KUKA KRL program: f1_Kuka_APT205T03S05.SRC

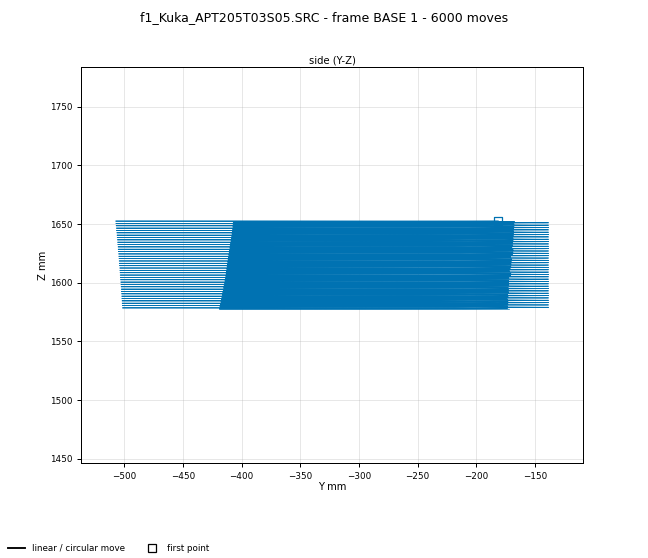
[picture p0: tool path of f1_Kuka_APT205T03S05.SRC in frame BASE 1, 6000 of 6001 moves have a stored position in this frame; points joined in program order, loops and branches not executed]
&ACCESS RVP
&REL 2
&PARAM TEMPLATE = C:\KRC\Roboter\Template\vorgabe
&PARAM EDITMASK = *
DEF f1_Kuka_APT205T03S05()


;FOLD INI;%{PE}%V3.2.0,%MKUKATPBASIS,%CINIT,%VCOMMON,%P
  ;FOLD BAS INI;%{E}%V3.2.0,%MKUKATPBASIS,%CINIT,%VINIT,%P
    GLOBAL INTERRUPT DECL 3 WHEN $STOPMESS==TRUE DO IR_STOPM ( )
    INTERRUPT ON 3
    BAS (#INITMOV,0 )
  ;ENDFOLD (BAS INI)
  ;FOLD USER INI;%{E}%V3.2.0,%MKUKATPUSER,%CINIT,%VINIT,%P
    ;Make your modifications here
  ;ENDFOLD (USER INI)
;ENDFOLD (INI)


;*** Make Null PTP Move
  PTP $pos_act

;*** Auto Load The Correct TOOL Data
  $tool=tool_data[3]

;*** Auto Load The Correct BASE Data
  $base=base_data[1]

  $ADVANCE = 5

;*** Restate Last Velocity
MMPM(30000.0)
SetRPM(6000)
LIN {X -0.097,Y -181.135,Z 1652.752,A 0.000,B 0.000,C 90.000,E1 135.405} C_DIS
LIN {X 0.030,Y -186.585,Z 1652.733,A 0.000,B 0.000,C 90.000,E1 132.000} C_DIS
LIN {X -0.021,Y -191.197,Z 1652.719,A 0.000,B 0.000,C 90.000,E1 129.519} C_DIS
LIN {X 0.024,Y -197.007,Z 1652.701,A 0.000,B 0.000,C 90.000,E1 126.217} C_DIS
LIN {X -0.058,Y -200.276,Z 1652.692,A 0.000,B 0.000,C 90.000,E1 124.612} C_DIS
LIN {X 0.005,Y -207.052,Z 1652.672,A 0.000,B 0.000,C 90.000,E1 120.924} C_DIS
LIN {X -0.045,Y -328.099,Z 1652.672,A 0.000,B 0.000,C 90.000,E1 120.924} C_DIS
LIN {X -0.152,Y -329.288,Z 1652.672,A 0.000,B 0.000,C 90.000,E1 120.924} C_DIS
LIN {X 0.100,Y -333.426,Z 1652.671,A 0.000,B 0.000,C 90.000,E1 120.718} C_DIS
LIN {X -0.104,Y -335.740,Z 1652.670,A 0.000,B 0.000,C 90.000,E1 120.590} C_DIS
LIN {X 0.166,Y -339.608,Z 1652.667,A 0.000,B 0.000,C 90.000,E1 120.129} C_DIS
LIN {X -0.040,Y -341.484,Z 1652.666,A 0.000,B 0.000,C 90.000,E1 119.873} C_DIS
LIN {X -0.079,Y -342.956,Z 1652.664,A 0.000,B 0.000,C 90.000,E1 119.589} C_DIS
LIN {X 0.037,Y -355.225,Z 1652.649,A 0.000,B 0.000,C 90.000,E1 116.821} C_DIS
LIN {X 0.029,Y -368.954,Z 1652.634,A 0.000,B 0.000,C 90.000,E1 114.131} C_DIS
LIN {X 0.163,Y -382.488,Z 1652.621,A 0.000,B 0.000,C 90.000,E1 111.770} C_DIS
LIN {X -0.003,Y -397.372,Z 1652.608,A 0.000,B 0.000,C 90.000,E1 109.504} C_DIS
LIN {X -0.071,Y -413.709,Z 1652.596,A 0.000,B 0.000,C 90.000,E1 107.275} C_DIS
LIN {X 0.146,Y -431.611,Z 1652.584,A 0.000,B 0.000,C 90.000,E1 105.064} C_DIS
LIN {X 0.171,Y -451.069,Z 1652.572,A 0.000,B 0.000,C 90.000,E1 102.952} C_DIS
LIN {X 0.102,Y -471.266,Z 1652.561,A 0.000,B 0.000,C 90.000,E1 101.007} C_DIS
LIN {X -0.176,Y -494.592,Z 1652.550,A 0.000,B 0.000,C 90.000,E1 99.029} C_DIS
LIN {X 0.166,Y -499.819,Z 1652.548,A 0.000,B 0.000,C 90.000,E1 98.568} C_DIS
LIN {X -0.174,Y -501.889,Z 1652.547,A 0.000,B 0.000,C 90.000,E1 98.398} C_DIS
LIN {X -0.238,Y -503.694,Z 1652.545,A 0.000,B 0.000,C 90.000,E1 98.163} C_DIS
LIN {X 0.198,Y -505.046,Z 1652.544,A 0.000,B 0.000,C 90.000,E1 97.871} C_DIS
LIN {X 0.003,Y -506.730,Z 1652.541,A 0.000,B 0.000,C 90.000,E1 97.409} C_DIS
LIN {X -0.185,Y -507.309,Z 1652.538,A 0.000,B 0.000,C 90.000,E1 96.947} C_DIS
LIN {X 0.141,Y -506.879,Z 1652.536,A 0.000,B 0.000,C 90.000,E1 96.429} C_DIS
LIN {X -0.035,Y -505.372,Z 1652.533,A 0.000,B 0.000,C 90.000,E1 95.967} C_DIS
LIN {X -0.149,Y -504.130,Z 1652.532,A 0.000,B 0.000,C 90.000,E1 95.739} C_DIS
LIN {X 0.200,Y -493.883,Z 1652.524,A 0.000,B 0.000,C 90.000,E1 94.245} C_DIS
LIN {X 0.044,Y -479.975,Z 1652.513,A 0.000,B 0.000,C 90.000,E1 92.293} C_DIS
LIN {X -0.050,Y -469.373,Z 1652.504,A 0.000,B 0.000,C 90.000,E1 90.802} C_DIS
LIN {X 0.134,Y -458.498,Z 1652.496,A 0.000,B 0.000,C 90.000,E1 89.255} C_DIS
LIN {X 0.134,Y -447.360,Z 1652.487,A 0.000,B 0.000,C 90.000,E1 87.707} C_DIS
LIN {X 0.215,Y -437.747,Z 1652.480,A 0.000,B 0.000,C 90.000,E1 86.388} C_DIS
LIN {X 0.171,Y -422.149,Z 1652.468,A 0.000,B 0.000,C 90.000,E1 84.261} C_DIS
LIN {X 0.124,Y -401.321,Z 1652.452,A 0.000,B 0.000,C 90.000,E1 81.254} C_DIS
LIN {X -0.095,Y -383.647,Z 1652.436,A 0.000,B 0.000,C 90.000,E1 78.465} C_DIS
LIN {X 0.146,Y -370.170,Z 1652.423,A 0.000,B 0.000,C 90.000,E1 76.117} C_DIS
LIN {X -0.154,Y -355.532,Z 1652.408,A 0.000,B 0.000,C 90.000,E1 73.504} C_DIS
LIN {X 0.037,Y -338.619,Z 1652.390,A 0.000,B 0.000,C 90.000,E1 70.134} C_DIS
LIN {X -0.145,Y -324.106,Z 1652.372,A 0.000,B 0.000,C 90.000,E1 67.050} C_DIS
LIN {X 0.007,Y -311.770,Z 1652.356,A 0.000,B 0.000,C 90.000,E1 64.152} C_DIS
LIN {X -0.105,Y -302.362,Z 1652.344,A 0.000,B 0.000,C 90.000,E1 61.897} C_DIS
LIN {X 0.124,Y -294.176,Z 1652.333,A 0.000,B 0.000,C 90.000,E1 59.871} C_DIS
LIN {X 0.086,Y -285.764,Z 1652.322,A 0.000,B 0.000,C 90.000,E1 57.867} C_DIS
LIN {X -0.036,Y -277.148,Z 1652.310,A 0.000,B 0.000,C 90.000,E1 55.849} C_DIS
LIN {X -0.016,Y -264.307,Z 1652.293,A 0.000,B 0.000,C 90.000,E1 52.718} C_DIS
LIN {X -0.141,Y -252.123,Z 1652.275,A 0.000,B 0.000,C 90.000,E1 49.542} C_DIS
LIN {X 0.060,Y -240.802,Z 1652.257,A 0.000,B 0.000,C 90.000,E1 46.215} C_DIS
LIN {X 0.093,Y -230.192,Z 1652.238,A 0.000,B 0.000,C 90.000,E1 42.852} C_DIS
LIN {X -0.001,Y -222.452,Z 1652.223,A 0.000,B 0.000,C 90.000,E1 40.216} C_DIS
LIN {X -0.092,Y -214.265,Z 1652.206,A 0.000,B 0.000,C 90.000,E1 37.156} C_DIS
LIN {X 0.005,Y -206.781,Z 1652.189,A 0.000,B 0.000,C 90.000,E1 33.992} C_DIS
LIN {X 0.029,Y -199.997,Z 1652.171,A 0.000,B 0.000,C 90.000,E1 30.797} C_DIS
LIN {X -0.070,Y -193.846,Z 1652.153,A 0.000,B 0.000,C 90.000,E1 27.590} C_DIS
LIN {X 0.025,Y -188.349,Z 1652.135,A 0.000,B 0.000,C 90.000,E1 24.283} C_DIS
LIN {X -0.004,Y -183.536,Z 1652.116,A 0.000,B 0.000,C 90.000,E1 20.972} C_DIS
LIN {X -0.072,Y -179.472,Z 1652.098,A 0.000,B 0.000,C 90.000,E1 17.638} C_DIS
LIN {X 0.069,Y -175.312,Z 1652.074,A 0.000,B 0.000,C 90.000,E1 13.355} C_DIS
LIN {X 0.019,Y -172.038,Z 1652.051,A 0.000,B 0.000,C 90.000,E1 9.095} C_DIS
LIN {X -0.078,Y -169.188,Z 1652.022,A 0.000,B 0.000,C 90.000,E1 3.955} C_DIS
LIN {X 0.014,Y -167.305,Z 1651.973,A 0.000,B 0.000,C 90.000,E1 355.179} C_DIS
LIN {X 0.071,Y -169.078,Z 1651.925,A 0.000,B 0.000,C 90.000,E1 346.464} C_DIS
LIN {X 0.068,Y -172.238,Z 1651.896,A 0.000,B 0.000,C 90.000,E1 341.275} C_DIS
LIN {X 0.041,Y -175.362,Z 1651.877,A 0.000,B 0.000,C 90.000,E1 337.847} C_DIS
LIN {X -0.036,Y -179.335,Z 1651.858,A 0.000,B 0.000,C 90.000,E1 334.460} C_DIS
LIN {X 0.059,Y -184.118,Z 1651.839,A 0.000,B 0.000,C 90.000,E1 331.051} C_DIS
LIN {X -0.040,Y -189.726,Z 1651.821,A 0.000,B 0.000,C 90.000,E1 327.740} C_DIS
LIN {X -0.042,Y -194.546,Z 1651.807,A 0.000,B 0.000,C 90.000,E1 325.261} C_DIS
LIN {X 0.008,Y -201.907,Z 1651.789,A 0.000,B 0.000,C 90.000,E1 321.984} C_DIS
LIN {X 0.018,Y -209.147,Z 1651.773,A 0.000,B 0.000,C 90.000,E1 319.175} C_DIS
LIN {X -0.091,Y -218.598,Z 1651.756,A 0.000,B 0.000,C 90.000,E1 316.053} C_DIS
LIN {X -0.050,Y -227.911,Z 1651.741,A 0.000,B 0.000,C 90.000,E1 313.338} C_DIS
LIN {X 0.015,Y -239.781,Z 1651.724,A 0.000,B 0.000,C 90.000,E1 310.297} C_DIS
LIN {X -0.068,Y -249.776,Z 1651.712,A 0.000,B 0.000,C 90.000,E1 308.096} C_DIS
LIN {X -0.143,Y -259.013,Z 1651.701,A 0.000,B 0.000,C 90.000,E1 306.297} C_DIS
LIN {X -0.036,Y -273.256,Z 1651.688,A 0.000,B 0.000,C 90.000,E1 303.785} C_DIS
LIN {X 0.115,Y -288.938,Z 1651.674,A 0.000,B 0.000,C 90.000,E1 301.337} C_DIS
LIN {X -0.030,Y -310.825,Z 1651.657,A 0.000,B 0.000,C 90.000,E1 298.359} C_DIS
LIN {X 0.020,Y -320.884,Z 1651.650,A 0.000,B 0.000,C 90.000,E1 297.052} C_DIS
LIN {X -0.030,Y -335.600,Z 1651.640,A 0.000,B 0.000,C 90.000,E1 295.155} C_DIS
LIN {X 0.067,Y -350.105,Z 1651.629,A 0.000,B 0.000,C 90.000,E1 293.281} C_DIS
LIN {X 0.115,Y -364.580,Z 1651.619,A 0.000,B 0.000,C 90.000,E1 291.461} C_DIS
LIN {X -0.048,Y -374.011,Z 1651.613,A 0.000,B 0.000,C 90.000,E1 290.301} C_DIS
LIN {X 0.143,Y -380.575,Z 1651.608,A 0.000,B 0.000,C 90.000,E1 289.396} C_DIS
LIN {X 0.032,Y -386.692,Z 1651.603,A 0.000,B 0.000,C 90.000,E1 288.544} C_DIS
LIN {X -0.020,Y -392.189,Z 1651.598,A 0.000,B 0.000,C 90.000,E1 287.692} C_DIS
LIN {X -0.150,Y -396.893,Z 1651.594,A 0.000,B 0.000,C 90.000,E1 286.858} C_DIS
LIN {X 0.156,Y -400.685,Z 1651.589,A 0.000,B 0.000,C 90.000,E1 285.969} C_DIS
LIN {X 0.110,Y -403.624,Z 1651.584,A 0.000,B 0.000,C 90.000,E1 285.134} C_DIS
LIN {X -0.006,Y -405.122,Z 1651.581,A 0.000,B 0.000,C 90.000,E1 284.592} C_DIS
LIN {X 0.179,Y -406.217,Z 1651.578,A 0.000,B 0.000,C 90.000,E1 284.008} C_DIS
LIN {X -0.019,Y -406.894,Z 1651.575,A 0.000,B 0.000,C 90.000,E1 283.480} C_DIS
LIN {X -0.117,Y -407.125,Z 1651.572,A 0.000,B 0.000,C 90.000,E1 282.939} C_DIS
LIN {X 0.090,Y -406.897,Z 1651.569,A 0.000,B 0.000,C 90.000,E1 282.355} C_DIS
LIN {X -0.096,Y -406.155,Z 1651.566,A 0.000,B 0.000,C 90.000,E1 281.827} C_DIS
LIN {X 0.112,Y -404.870,Z 1651.563,A 0.000,B 0.000,C 90.000,E1 281.243} C_DIS
LIN {X -0.082,Y -403.014,Z 1651.559,A 0.000,B 0.000,C 90.000,E1 280.715} C_DIS
LIN {X 0.041,Y -400.509,Z 1651.556,A 0.000,B 0.000,C 90.000,E1 280.141} C_DIS
LIN {X -0.175,Y -397.400,Z 1651.553,A 0.000,B 0.000,C 90.000,E1 279.613} C_DIS
LIN {X -0.013,Y -391.663,Z 1651.549,A 0.000,B 0.000,C 90.000,E1 278.746} C_DIS
LIN {X 0.157,Y -385.162,Z 1651.544,A 0.000,B 0.000,C 90.000,E1 277.871} C_DIS
LIN {X 0.179,Y -380.478,Z 1651.541,A 0.000,B 0.000,C 90.000,E1 277.296} C_DIS
LIN {X 0.178,Y -375.244,Z 1651.537,A 0.000,B 0.000,C 90.000,E1 276.720} C_DIS
LIN {X -0.092,Y -369.505,Z 1651.534,A 0.000,B 0.000,C 90.000,E1 276.201} C_DIS
LIN {X -0.088,Y -363.404,Z 1651.531,A 0.000,B 0.000,C 90.000,E1 275.682} C_DIS
LIN {X -0.133,Y -357.073,Z 1651.529,A 0.000,B 0.000,C 90.000,E1 275.220} C_DIS
LIN {X 0.049,Y -347.576,Z 1651.526,A 0.000,B 0.000,C 90.000,E1 274.588} C_DIS
LIN {X -0.095,Y -338.016,Z 1651.523,A 0.000,B 0.000,C 90.000,E1 274.073} C_DIS
LIN {X 0.074,Y -328.401,Z 1651.520,A 0.000,B 0.000,C 90.000,E1 273.555} C_DIS
LIN {X 0.143,Y -318.459,Z 1651.517,A 0.000,B 0.000,C 90.000,E1 273.094} C_DIS
LIN {X -0.120,Y -308.289,Z 1651.515,A 0.000,B 0.000,C 90.000,E1 272.751} C_DIS
LIN {X -0.106,Y -301.207,Z 1651.514,A 0.000,B 0.000,C 90.000,E1 272.522} C_DIS
LIN {X -0.076,Y -290.309,Z 1651.512,A 0.000,B 0.000,C 90.000,E1 272.236} C_DIS
LIN {X -0.004,Y -282.504,Z 1651.511,A 0.000,B 0.000,C 90.000,E1 272.064} C_DIS
LIN {X -0.082,Y -272.258,Z 1651.511,A 0.000,B 0.000,C 90.000,E1 271.949} C_DIS
LIN {X -0.062,Y -240.164,Z 1651.510,A 0.000,B 0.000,C 90.000,E1 271.718} C_DIS
LIN {X 0.010,Y -211.026,Z 1651.509,A 0.000,B 0.000,C 90.000,E1 271.547} C_DIS
LIN {X 0.094,Y -186.358,Z 1651.508,A 0.000,B 0.000,C 90.000,E1 271.432} C_DIS
LIN {X 0.060,Y -181.360,Z 1651.508,A 0.000,B 0.000,C 90.000,E1 271.432} C_DIS
LIN {X -0.034,Y -181.556,Z 1651.503,A 0.000,B 0.000,C 90.000,E1 270.573} C_DIS
LIN {X 0.076,Y -181.292,Z 1651.494,A 0.000,B 0.000,C 90.000,E1 268.854} C_DIS
LIN {X -0.055,Y -180.907,Z 1651.475,A 0.000,B 0.000,C 90.000,E1 265.527} C_DIS
LIN {X 0.003,Y -180.754,Z 1651.470,A 0.000,B 0.000,C 90.000,E1 264.666} C_DIS
LIN {X 0.070,Y -178.846,Z 1651.442,A 0.000,B 0.000,C 90.000,E1 259.577} C_DIS
LIN {X -0.033,Y -175.890,Z 1651.414,A 0.000,B 0.000,C 90.000,E1 254.519} C_DIS
LIN {X 0.072,Y -174.560,Z 1651.404,A 0.000,B 0.000,C 90.000,E1 252.779} C_DIS
LIN {X -0.058,Y -171.544,Z 1651.381,A 0.000,B 0.000,C 90.000,E1 248.539} C_DIS
LIN {X -0.002,Y -167.768,Z 1651.357,A 0.000,B 0.000,C 90.000,E1 244.204} C_DIS
LIN {X -0.061,Y -166.477,Z 1651.347,A 0.000,B 0.000,C 90.000,E1 242.487} C_DIS
LIN {X -0.064,Y -163.189,Z 1651.328,A 0.000,B 0.000,C 90.000,E1 238.997} C_DIS
LIN {X -0.009,Y -161.152,Z 1651.313,A 0.000,B 0.000,C 90.000,E1 236.342} C_DIS
LIN {X 0.026,Y -157.169,Z 1651.288,A 0.000,B 0.000,C 90.000,E1 231.904} C_DIS
LIN {X -0.051,Y -155.901,Z 1651.279,A 0.000,B 0.000,C 90.000,E1 230.150} C_DIS
LIN {X 0.007,Y -152.151,Z 1651.254,A 0.000,B 0.000,C 90.000,E1 225.648} C_DIS
LIN {X 0.027,Y -150.400,Z 1651.239,A 0.000,B 0.000,C 90.000,E1 222.933} C_DIS
LIN {X 0.050,Y -147.130,Z 1651.213,A 0.000,B 0.000,C 90.000,E1 218.382} C_DIS
LIN {X -0.044,Y -145.692,Z 1651.198,A 0.000,B 0.000,C 90.000,E1 215.678} C_DIS
LIN {X 0.038,Y -143.074,Z 1651.173,A 0.000,B 0.000,C 90.000,E1 211.052} C_DIS
LIN {X -0.031,Y -141.694,Z 1651.152,A 0.000,B 0.000,C 90.000,E1 207.385} C_DIS
LIN {X 0.023,Y -139.464,Z 1651.116,A 0.000,B 0.000,C 90.000,E1 200.865} C_DIS
LIN {X -0.053,Y -139.197,Z 1651.106,A 0.000,B 0.000,C 90.000,E1 199.033} C_DIS
LIN {X 0.010,Y -138.326,Z 1651.054,A 0.000,B 0.000,C 90.000,E1 189.670} C_DIS
LIN {X 0.015,Y -139.449,Z 1651.007,A 0.000,B 0.000,C 90.000,E1 181.260} C_DIS
LIN {X -0.045,Y -140.991,Z 1650.976,A 0.000,B 0.000,C 90.000,E1 175.698} C_DIS
LIN {X 0.046,Y -142.746,Z 1650.955,A 0.000,B 0.000,C 90.000,E1 171.951} C_DIS
LIN {X 0.003,Y -145.142,Z 1650.930,A 0.000,B 0.000,C 90.000,E1 167.353} C_DIS
LIN {X -0.005,Y -147.765,Z 1650.909,A 0.000,B 0.000,C 90.000,E1 163.685} C_DIS
LIN {X -0.065,Y -150.438,Z 1650.889,A 0.000,B 0.000,C 90.000,E1 160.061} C_DIS
LIN {X 0.010,Y -153.883,Z 1650.869,A 0.000,B 0.000,C 90.000,E1 156.410} C_DIS
LIN {X 0.005,Y -157.294,Z 1650.849,A 0.000,B 0.000,C 90.000,E1 152.820} C_DIS
LIN {X -0.059,Y -161.477,Z 1650.829,A 0.000,B 0.000,C 90.000,E1 149.282} C_DIS
LIN {X 0.040,Y -165.676,Z 1650.810,A 0.000,B 0.000,C 90.000,E1 145.722} C_DIS
LIN {X -0.073,Y -170.616,Z 1650.790,A 0.000,B 0.000,C 90.000,E1 142.271} C_DIS
LIN {X 0.081,Y -175.493,Z 1650.771,A 0.000,B 0.000,C 90.000,E1 138.771} C_DIS
LIN {X -0.053,Y -181.115,Z 1650.752,A 0.000,B 0.000,C 90.000,E1 135.405} C_DIS
LIN {X 0.075,Y -186.560,Z 1650.734,A 0.000,B 0.000,C 90.000,E1 132.000} C_DIS
LIN {X 0.025,Y -191.175,Z 1650.720,A 0.000,B 0.000,C 90.000,E1 129.519} C_DIS
LIN {X 0.071,Y -196.980,Z 1650.701,A 0.000,B 0.000,C 90.000,E1 126.217} C_DIS
LIN {X -0.010,Y -200.248,Z 1650.692,A 0.000,B 0.000,C 90.000,E1 124.612} C_DIS
LIN {X -0.120,Y -206.964,Z 1650.672,A 0.000,B 0.000,C 90.000,E1 121.003} C_DIS
LIN {X 0.200,Y -327.654,Z 1650.672,A 0.000,B 0.000,C 90.000,E1 120.924} C_DIS
LIN {X 0.141,Y -328.515,Z 1650.672,A 0.000,B 0.000,C 90.000,E1 120.924} C_DIS
LIN {X -0.171,Y -333.376,Z 1650.671,A 0.000,B 0.000,C 90.000,E1 120.797} C_DIS
LIN {X -0.026,Y -335.871,Z 1650.670,A 0.000,B 0.000,C 90.000,E1 120.590} C_DIS
LIN {X 0.171,Y -339.702,Z 1650.668,A 0.000,B 0.000,C 90.000,E1 120.129} C_DIS
LIN {X -0.083,Y -341.558,Z 1650.666,A 0.000,B 0.000,C 90.000,E1 119.873} C_DIS
LIN {X -0.183,Y -344.305,Z 1650.662,A 0.000,B 0.000,C 90.000,E1 119.283} C_DIS
LIN {X 0.136,Y -356.727,Z 1650.647,A 0.000,B 0.000,C 90.000,E1 116.488} C_DIS
LIN {X 0.019,Y -370.631,Z 1650.632,A 0.000,B 0.000,C 90.000,E1 113.823} C_DIS
LIN {X 0.058,Y -384.336,Z 1650.619,A 0.000,B 0.000,C 90.000,E1 111.482} C_DIS
LIN {X -0.054,Y -399.404,Z 1650.607,A 0.000,B 0.000,C 90.000,E1 109.214} C_DIS
LIN {X -0.062,Y -415.939,Z 1650.594,A 0.000,B 0.000,C 90.000,E1 106.985} C_DIS
LIN {X 0.219,Y -434.054,Z 1650.582,A 0.000,B 0.000,C 90.000,E1 104.773} C_DIS
LIN {X 0.044,Y -453.650,Z 1650.571,A 0.000,B 0.000,C 90.000,E1 102.703} C_DIS
LIN {X -0.051,Y -473.919,Z 1650.560,A 0.000,B 0.000,C 90.000,E1 100.782} C_DIS
LIN {X 0.070,Y -499.894,Z 1650.548,A 0.000,B 0.000,C 90.000,E1 98.568} C_DIS
LIN {X -0.271,Y -501.898,Z 1650.547,A 0.000,B 0.000,C 90.000,E1 98.398} C_DIS
LIN {X 0.156,Y -503.659,Z 1650.545,A 0.000,B 0.000,C 90.000,E1 98.106} C_DIS
LIN {X 0.085,Y -504.975,Z 1650.544,A 0.000,B 0.000,C 90.000,E1 97.871} C_DIS
LIN {X -0.111,Y -506.596,Z 1650.541,A 0.000,B 0.000,C 90.000,E1 97.409} C_DIS
LIN {X 0.204,Y -507.121,Z 1650.538,A 0.000,B 0.000,C 90.000,E1 96.891} C_DIS
LIN {X 0.025,Y -506.639,Z 1650.536,A 0.000,B 0.000,C 90.000,E1 96.429} C_DIS
LIN {X -0.150,Y -505.071,Z 1650.533,A 0.000,B 0.000,C 90.000,E1 95.967} C_DIS
LIN {X 0.237,Y -503.791,Z 1650.532,A 0.000,B 0.000,C 90.000,E1 95.682} C_DIS
LIN {X 0.081,Y -493.527,Z 1650.524,A 0.000,B 0.000,C 90.000,E1 94.245} C_DIS
LIN {X 0.086,Y -481.406,Z 1650.514,A 0.000,B 0.000,C 90.000,E1 92.522} C_DIS
LIN {X 0.014,Y -470.855,Z 1650.506,A 0.000,B 0.000,C 90.000,E1 91.031} C_DIS
LIN {X 0.221,Y -460.025,Z 1650.497,A 0.000,B 0.000,C 90.000,E1 89.484} C_DIS
LIN {X -0.202,Y -448.922,Z 1650.489,A 0.000,B 0.000,C 90.000,E1 87.993} C_DIS
LIN {X 0.083,Y -437.388,Z 1650.480,A 0.000,B 0.000,C 90.000,E1 86.388} C_DIS
LIN {X 0.035,Y -421.766,Z 1650.468,A 0.000,B 0.000,C 90.000,E1 84.261} C_DIS
LIN {X -0.113,Y -402.770,Z 1650.453,A 0.000,B 0.000,C 90.000,E1 81.546} C_DIS
LIN {X 0.095,Y -384.990,Z 1650.437,A 0.000,B 0.000,C 90.000,E1 78.701} C_DIS
LIN {X -0.005,Y -369.796,Z 1650.423,A 0.000,B 0.000,C 90.000,E1 76.117} C_DIS
LIN {X 0.076,Y -353.593,Z 1650.406,A 0.000,B 0.000,C 90.000,E1 73.142} C_DIS
LIN {X -0.120,Y -336.788,Z 1650.388,A 0.000,B 0.000,C 90.000,E1 69.826} C_DIS
LIN {X 0.027,Y -320.966,Z 1650.369,A 0.000,B 0.000,C 90.000,E1 66.357} C_DIS
LIN {X 0.084,Y -308.749,Z 1650.353,A 0.000,B 0.000,C 90.000,E1 63.461} C_DIS
LIN {X 0.044,Y -299.319,Z 1650.340,A 0.000,B 0.000,C 90.000,E1 61.179} C_DIS
LIN {X -0.043,Y -291.088,Z 1650.329,A 0.000,B 0.000,C 90.000,E1 59.203} C_DIS
LIN {X 0.018,Y -282.620,Z 1650.318,A 0.000,B 0.000,C 90.000,E1 57.168} C_DIS
LIN {X 0.015,Y -272.476,Z 1650.304,A 0.000,B 0.000,C 90.000,E1 54.769} C_DIS
LIN {X -0.060,Y -261.263,Z 1650.289,A 0.000,B 0.000,C 90.000,E1 51.984} C_DIS
LIN {X -0.101,Y -249.276,Z 1650.271,A 0.000,B 0.000,C 90.000,E1 48.771} C_DIS
LIN {X 0.018,Y -238.112,Z 1650.252,A 0.000,B 0.000,C 90.000,E1 45.445} C_DIS
LIN {X -0.017,Y -227.619,Z 1650.234,A 0.000,B 0.000,C 90.000,E1 42.081} C_DIS
LIN {X 0.044,Y -217.954,Z 1650.215,A 0.000,B 0.000,C 90.000,E1 38.624} C_DIS
LIN {X 0.016,Y -210.146,Z 1650.197,A 0.000,B 0.000,C 90.000,E1 35.518} C_DIS
LIN {X 0.060,Y -203.018,Z 1650.180,A 0.000,B 0.000,C 90.000,E1 32.339} C_DIS
LIN {X -0.045,Y -196.623,Z 1650.162,A 0.000,B 0.000,C 90.000,E1 29.155} C_DIS
LIN {X -0.056,Y -190.802,Z 1650.144,A 0.000,B 0.000,C 90.000,E1 25.899} C_DIS
LIN {X -0.026,Y -185.727,Z 1650.125,A 0.000,B 0.000,C 90.000,E1 22.589} C_DIS
LIN {X -0.085,Y -181.303,Z 1650.107,A 0.000,B 0.000,C 90.000,E1 19.268} C_DIS
LIN {X 0.039,Y -176.851,Z 1650.083,A 0.000,B 0.000,C 90.000,E1 15.009} C_DIS
LIN {X -0.067,Y -173.246,Z 1650.060,A 0.000,B 0.000,C 90.000,E1 10.782} C_DIS
LIN {X -0.072,Y -170.026,Z 1650.031,A 0.000,B 0.000,C 90.000,E1 5.625} C_DIS
LIN {X -0.059,Y -167.699,Z 1649.993,A 0.000,B 0.000,C 90.000,E1 358.682} C_DIS
LIN {X 0.014,Y -168.784,Z 1649.930,A 0.000,B 0.000,C 90.000,E1 347.353} C_DIS
LIN {X -0.054,Y -171.693,Z 1649.901,A 0.000,B 0.000,C 90.000,E1 342.181} C_DIS
LIN {X 0.005,Y -174.600,Z 1649.882,A 0.000,B 0.000,C 90.000,E1 338.720} C_DIS
LIN {X -0.004,Y -178.380,Z 1649.863,A 0.000,B 0.000,C 90.000,E1 335.305} C_DIS
LIN {X 0.061,Y -182.998,Z 1649.844,A 0.000,B 0.000,C 90.000,E1 331.897} C_DIS
LIN {X 0.100,Y -188.435,Z 1649.825,A 0.000,B 0.000,C 90.000,E1 328.535} C_DIS
LIN {X -0.025,Y -193.049,Z 1649.812,A 0.000,B 0.000,C 90.000,E1 326.087} C_DIS
LIN {X -0.010,Y -198.301,Z 1649.798,A 0.000,B 0.000,C 90.000,E1 323.623} C_DIS
LIN {X 0.103,Y -206.105,Z 1649.780,A 0.000,B 0.000,C 90.000,E1 320.356} C_DIS
LIN {X -0.103,Y -213.901,Z 1649.765,A 0.000,B 0.000,C 90.000,E1 317.634} C_DIS
LIN {X -0.018,Y -222.623,Z 1649.749,A 0.000,B 0.000,C 90.000,E1 314.879} C_DIS
LIN {X -0.043,Y -232.353,Z 1649.734,A 0.000,B 0.000,C 90.000,E1 312.204} C_DIS
LIN {X 0.038,Y -241.461,Z 1649.722,A 0.000,B 0.000,C 90.000,E1 309.930} C_DIS
LIN {X -0.010,Y -251.633,Z 1649.710,A 0.000,B 0.000,C 90.000,E1 307.729} C_DIS
LIN {X -0.061,Y -261.015,Z 1649.700,A 0.000,B 0.000,C 90.000,E1 305.931} C_DIS
LIN {X 0.027,Y -277.617,Z 1649.684,A 0.000,B 0.000,C 90.000,E1 303.086} C_DIS
LIN {X 0.112,Y -296.057,Z 1649.669,A 0.000,B 0.000,C 90.000,E1 300.335} C_DIS
LIN {X -0.025,Y -315.928,Z 1649.654,A 0.000,B 0.000,C 90.000,E1 297.719} C_DIS
LIN {X 0.035,Y -328.266,Z 1649.645,A 0.000,B 0.000,C 90.000,E1 296.104} C_DIS
LIN {X 0.140,Y -340.445,Z 1649.636,A 0.000,B 0.000,C 90.000,E1 294.515} C_DIS
LIN {X 0.007,Y -354.935,Z 1649.626,A 0.000,B 0.000,C 90.000,E1 292.695} C_DIS
LIN {X -0.209,Y -366.952,Z 1649.618,A 0.000,B 0.000,C 90.000,E1 291.227} C_DIS
LIN {X 0.134,Y -376.208,Z 1649.611,A 0.000,B 0.000,C 90.000,E1 289.993} C_DIS
LIN {X -0.018,Y -382.676,Z 1649.606,A 0.000,B 0.000,C 90.000,E1 289.141} C_DIS
LIN {X -0.109,Y -388.591,Z 1649.602,A 0.000,B 0.000,C 90.000,E1 288.290} C_DIS
LIN {X 0.100,Y -393.889,Z 1649.597,A 0.000,B 0.000,C 90.000,E1 287.402} C_DIS
LIN {X -0.064,Y -396.955,Z 1649.594,A 0.000,B 0.000,C 90.000,E1 286.858} C_DIS
LIN {X -0.142,Y -400.771,Z 1649.589,A 0.000,B 0.000,C 90.000,E1 286.024} C_DIS
LIN {X -0.190,Y -403.699,Z 1649.584,A 0.000,B 0.000,C 90.000,E1 285.190} C_DIS
LIN {X 0.084,Y -405.228,Z 1649.581,A 0.000,B 0.000,C 90.000,E1 284.592} C_DIS
LIN {X -0.125,Y -406.315,Z 1649.578,A 0.000,B 0.000,C 90.000,E1 284.064} C_DIS
LIN {X 0.073,Y -407.039,Z 1649.575,A 0.000,B 0.000,C 90.000,E1 283.480} C_DIS
LIN {X -0.026,Y -407.287,Z 1649.572,A 0.000,B 0.000,C 90.000,E1 282.939} C_DIS
LIN {X 0.183,Y -407.080,Z 1649.569,A 0.000,B 0.000,C 90.000,E1 282.355} C_DIS
LIN {X -0.004,Y -406.366,Z 1649.566,A 0.000,B 0.000,C 90.000,E1 281.827} C_DIS
LIN {X 0.207,Y -405.100,Z 1649.563,A 0.000,B 0.000,C 90.000,E1 281.243} C_DIS
LIN {X 0.013,Y -403.233,Z 1649.560,A 0.000,B 0.000,C 90.000,E1 280.715} C_DIS
LIN {X 0.137,Y -400.774,Z 1649.556,A 0.000,B 0.000,C 90.000,E1 280.141} C_DIS
LIN {X -0.079,Y -397.634,Z 1649.553,A 0.000,B 0.000,C 90.000,E1 279.613} C_DIS
LIN {X 0.084,Y -391.868,Z 1649.549,A 0.000,B 0.000,C 90.000,E1 278.746} C_DIS
LIN {X -0.140,Y -383.042,Z 1649.542,A 0.000,B 0.000,C 90.000,E1 277.644} C_DIS
LIN {X -0.116,Y -378.074,Z 1649.539,A 0.000,B 0.000,C 90.000,E1 277.068} C_DIS
LIN {X -0.011,Y -372.606,Z 1649.536,A 0.000,B 0.000,C 90.000,E1 276.486} C_DIS
LIN {X -0.137,Y -366.668,Z 1649.533,A 0.000,B 0.000,C 90.000,E1 275.967} C_DIS
LIN {X -0.020,Y -360.484,Z 1649.530,A 0.000,B 0.000,C 90.000,E1 275.454} C_DIS
LIN {X 0.077,Y -354.071,Z 1649.528,A 0.000,B 0.000,C 90.000,E1 274.992} C_DIS
LIN {X 0.020,Y -344.424,Z 1649.525,A 0.000,B 0.000,C 90.000,E1 274.416} C_DIS
LIN {X 0.015,Y -334.900,Z 1649.522,A 0.000,B 0.000,C 90.000,E1 273.898} C_DIS
LIN {X -0.103,Y -325.109,Z 1649.519,A 0.000,B 0.000,C 90.000,E1 273.440} C_DIS
LIN {X 0.098,Y -315.096,Z 1649.517,A 0.000,B 0.000,C 90.000,E1 272.980} C_DIS
LIN {X -0.025,Y -304.909,Z 1649.515,A 0.000,B 0.000,C 90.000,E1 272.636} C_DIS
LIN {X -0.089,Y -294.291,Z 1649.513,A 0.000,B 0.000,C 90.000,E1 272.350} C_DIS
LIN {X -0.074,Y -286.938,Z 1649.512,A 0.000,B 0.000,C 90.000,E1 272.178} C_DIS
LIN {X 0.062,Y -278.543,Z 1649.511,A 0.000,B 0.000,C 90.000,E1 272.007} C_DIS
LIN {X -0.073,Y -262.554,Z 1649.510,A 0.000,B 0.000,C 90.000,E1 271.892} C_DIS
LIN {X 0.060,Y -233.163,Z 1649.509,A 0.000,B 0.000,C 90.000,E1 271.661} C_DIS
LIN {X 0.064,Y -211.839,Z 1649.509,A 0.000,B 0.000,C 90.000,E1 271.547} C_DIS
LIN {X -0.046,Y -183.974,Z 1649.508,A 0.000,B 0.000,C 90.000,E1 271.489} C_DIS
LIN {X -0.075,Y -181.357,Z 1649.508,A 0.000,B 0.000,C 90.000,E1 271.489} C_DIS
LIN {X 0.011,Y -181.553,Z 1649.503,A 0.000,B 0.000,C 90.000,E1 270.573} C_DIS
LIN {X -0.061,Y -181.295,Z 1649.494,A 0.000,B 0.000,C 90.000,E1 268.912} C_DIS
LIN {X -0.011,Y -180.907,Z 1649.475,A 0.000,B 0.000,C 90.000,E1 265.527} C_DIS
LIN {X 0.046,Y -180.760,Z 1649.470,A 0.000,B 0.000,C 90.000,E1 264.666} C_DIS
LIN {X -0.062,Y -178.853,Z 1649.442,A 0.000,B 0.000,C 90.000,E1 259.634} C_DIS
LIN {X 0.010,Y -175.896,Z 1649.414,A 0.000,B 0.000,C 90.000,E1 254.519} C_DIS
LIN {X -0.051,Y -174.572,Z 1649.405,A 0.000,B 0.000,C 90.000,E1 252.834} C_DIS
LIN {X -0.015,Y -171.555,Z 1649.381,A 0.000,B 0.000,C 90.000,E1 248.539} C_DIS
LIN {X 0.040,Y -167.779,Z 1649.357,A 0.000,B 0.000,C 90.000,E1 244.204} C_DIS
LIN {X -0.019,Y -166.491,Z 1649.347,A 0.000,B 0.000,C 90.000,E1 242.487} C_DIS
LIN {X -0.023,Y -163.202,Z 1649.328,A 0.000,B 0.000,C 90.000,E1 238.997} C_DIS
LIN {X 0.031,Y -161.166,Z 1649.313,A 0.000,B 0.000,C 90.000,E1 236.342} C_DIS
LIN {X 0.067,Y -157.181,Z 1649.288,A 0.000,B 0.000,C 90.000,E1 231.904} C_DIS
LIN {X -0.010,Y -155.911,Z 1649.279,A 0.000,B 0.000,C 90.000,E1 230.150} C_DIS
LIN {X 0.046,Y -152.161,Z 1649.254,A 0.000,B 0.000,C 90.000,E1 225.648} C_DIS
LIN {X 0.066,Y -150.410,Z 1649.239,A 0.000,B 0.000,C 90.000,E1 222.933} C_DIS
LIN {X 0.088,Y -147.139,Z 1649.213,A 0.000,B 0.000,C 90.000,E1 218.382} C_DIS
LIN {X -0.006,Y -145.698,Z 1649.198,A 0.000,B 0.000,C 90.000,E1 215.678} C_DIS
LIN {X 0.002,Y -143.082,Z 1649.173,A 0.000,B 0.000,C 90.000,E1 211.082} C_DIS
LIN {X 0.008,Y -141.700,Z 1649.152,A 0.000,B 0.000,C 90.000,E1 207.385} C_DIS
LIN {X -0.070,Y -139.466,Z 1649.116,A 0.000,B 0.000,C 90.000,E1 200.918} C_DIS
LIN {X -0.016,Y -139.199,Z 1649.106,A 0.000,B 0.000,C 90.000,E1 199.033} C_DIS
LIN {X 0.048,Y -138.327,Z 1649.054,A 0.000,B 0.000,C 90.000,E1 189.670} C_DIS
LIN {X 0.053,Y -139.446,Z 1649.007,A 0.000,B 0.000,C 90.000,E1 181.260} C_DIS
LIN {X -0.007,Y -140.985,Z 1648.976,A 0.000,B 0.000,C 90.000,E1 175.698} C_DIS
LIN {X -0.057,Y -142.739,Z 1648.955,A 0.000,B 0.000,C 90.000,E1 172.008} C_DIS
LIN {X 0.040,Y -145.132,Z 1648.930,A 0.000,B 0.000,C 90.000,E1 167.353} C_DIS
LIN {X 0.035,Y -147.755,Z 1648.909,A 0.000,B 0.000,C 90.000,E1 163.685} C_DIS
LIN {X -0.026,Y -150.426,Z 1648.889,A 0.000,B 0.000,C 90.000,E1 160.061} C_DIS
LIN {X -0.011,Y -153.868,Z 1648.869,A 0.000,B 0.000,C 90.000,E1 156.433} C_DIS
LIN {X 0.045,Y -157.278,Z 1648.849,A 0.000,B 0.000,C 90.000,E1 152.820} C_DIS
LIN {X -0.018,Y -161.458,Z 1648.829,A 0.000,B 0.000,C 90.000,E1 149.282} C_DIS
LIN {X -0.012,Y -165.658,Z 1648.810,A 0.000,B 0.000,C 90.000,E1 145.754} C_DIS
LIN {X -0.030,Y -170.593,Z 1648.790,A 0.000,B 0.000,C 90.000,E1 142.271} C_DIS
LIN {X 0.009,Y -175.471,Z 1648.771,A 0.000,B 0.000,C 90.000,E1 138.809} C_DIS
LIN {X -0.009,Y -181.094,Z 1648.752,A 0.000,B 0.000,C 90.000,E1 135.405} C_DIS
LIN {X -0.019,Y -186.536,Z 1648.734,A 0.000,B 0.000,C 90.000,E1 132.043} C_DIS
LIN {X -0.077,Y -191.152,Z 1648.720,A 0.000,B 0.000,C 90.000,E1 129.564} C_DIS
LIN {X 0.001,Y -196.955,Z 1648.701,A 0.000,B 0.000,C 90.000,E1 126.251} C_DIS
LIN {X 0.037,Y -200.220,Z 1648.692,A 0.000,B 0.000,C 90.000,E1 124.612} C_DIS
LIN {X 0.004,Y -206.895,Z 1648.672,A 0.000,B 0.000,C 90.000,E1 121.003} C_DIS
LIN {X -0.053,Y -328.016,Z 1648.672,A 0.000,B 0.000,C 90.000,E1 121.003} C_DIS
LIN {X 0.219,Y -329.582,Z 1648.672,A 0.000,B 0.000,C 90.000,E1 120.924} C_DIS
LIN {X -0.092,Y -333.620,Z 1648.671,A 0.000,B 0.000,C 90.000,E1 120.797} C_DIS
LIN {X 0.051,Y -335.989,Z 1648.670,A 0.000,B 0.000,C 90.000,E1 120.590} C_DIS
LIN {X 0.135,Y -339.835,Z 1648.667,A 0.000,B 0.000,C 90.000,E1 120.129} C_DIS
LIN {X -0.171,Y -341.663,Z 1648.666,A 0.000,B 0.000,C 90.000,E1 119.873} C_DIS
LIN {X 0.002,Y -348.369,Z 1648.657,A 0.000,B 0.000,C 90.000,E1 118.309} C_DIS
LIN {X -0.032,Y -361.281,Z 1648.642,A 0.000,B 0.000,C 90.000,E1 115.591} C_DIS
LIN {X 0.158,Y -375.724,Z 1648.627,A 0.000,B 0.000,C 90.000,E1 112.898} C_DIS
LIN {X -0.027,Y -389.942,Z 1648.615,A 0.000,B 0.000,C 90.000,E1 110.610} C_DIS
LIN {X -0.145,Y -405.561,Z 1648.602,A 0.000,B 0.000,C 90.000,E1 108.362} C_DIS
LIN {X -0.012,Y -422.690,Z 1648.590,A 0.000,B 0.000,C 90.000,E1 106.134} C_DIS
LIN {X -0.218,Y -441.447,Z 1648.578,A 0.000,B 0.000,C 90.000,E1 104.008} C_DIS
LIN {X -0.053,Y -461.367,Z 1648.566,A 0.000,B 0.000,C 90.000,E1 101.951} C_DIS
LIN {X 0.018,Y -484.422,Z 1648.555,A 0.000,B 0.000,C 90.000,E1 99.849} C_DIS
LIN {X -0.073,Y -500.017,Z 1648.548,A 0.000,B 0.000,C 90.000,E1 98.568} C_DIS
LIN {X 0.084,Y -501.943,Z 1648.546,A 0.000,B 0.000,C 90.000,E1 98.341} C_DIS
LIN {X 0.015,Y -503.644,Z 1648.545,A 0.000,B 0.000,C 90.000,E1 98.106} C_DIS
LIN {X -0.058,Y -504.915,Z 1648.544,A 0.000,B 0.000,C 90.000,E1 97.871} C_DIS
LIN {X 0.248,Y -506.465,Z 1648.541,A 0.000,B 0.000,C 90.000,E1 97.352} C_DIS
LIN {X 0.060,Y -506.931,Z 1648.538,A 0.000,B 0.000,C 90.000,E1 96.891} C_DIS
LIN {X -0.119,Y -506.389,Z 1648.536,A 0.000,B 0.000,C 90.000,E1 96.429} C_DIS
LIN {X 0.207,Y -504.751,Z 1648.533,A 0.000,B 0.000,C 90.000,E1 95.910} C_DIS
LIN {X 0.092,Y -503.427,Z 1648.532,A 0.000,B 0.000,C 90.000,E1 95.682} C_DIS
LIN {X -0.068,Y -493.149,Z 1648.524,A 0.000,B 0.000,C 90.000,E1 94.245} C_DIS
LIN {X -0.066,Y -481.061,Z 1648.514,A 0.000,B 0.000,C 90.000,E1 92.522} C_DIS
LIN {X -0.139,Y -470.525,Z 1648.506,A 0.000,B 0.000,C 90.000,E1 91.031} C_DIS
LIN {X 0.066,Y -459.697,Z 1648.497,A 0.000,B 0.000,C 90.000,E1 89.484} C_DIS
LIN {X 0.090,Y -448.583,Z 1648.489,A 0.000,B 0.000,C 90.000,E1 87.936} C_DIS
LIN {X 0.186,Y -438.955,Z 1648.481,A 0.000,B 0.000,C 90.000,E1 86.617} C_DIS
LIN {X 0.016,Y -425.258,Z 1648.471,A 0.000,B 0.000,C 90.000,E1 84.780} C_DIS
LIN {X 0.140,Y -409.802,Z 1648.459,A 0.000,B 0.000,C 90.000,E1 82.591} C_DIS
LIN {X 0.216,Y -389.780,Z 1648.442,A 0.000,B 0.000,C 90.000,E1 79.511} C_DIS
LIN {X 0.172,Y -374.389,Z 1648.428,A 0.000,B 0.000,C 90.000,E1 76.937} C_DIS
LIN {X -0.113,Y -359.581,Z 1648.413,A 0.000,B 0.000,C 90.000,E1 74.338} C_DIS
LIN {X -0.141,Y -345.424,Z 1648.398,A 0.000,B 0.000,C 90.000,E1 71.638} C_DIS
LIN {X -0.020,Y -331.978,Z 1648.382,A 0.000,B 0.000,C 90.000,E1 68.847} C_DIS
LIN {X 0.153,Y -317.833,Z 1648.365,A 0.000,B 0.000,C 90.000,E1 65.665} C_DIS
LIN {X -0.062,Y -307.052,Z 1648.351,A 0.000,B 0.000,C 90.000,E1 63.127} C_DIS
LIN {X 0.115,Y -298.969,Z 1648.340,A 0.000,B 0.000,C 90.000,E1 61.129} C_DIS
LIN {X 0.015,Y -290.748,Z 1648.329,A 0.000,B 0.000,C 90.000,E1 59.154} C_DIS
LIN {X 0.063,Y -282.290,Z 1648.317,A 0.000,B 0.000,C 90.000,E1 57.120} C_DIS
LIN {X -0.120,Y -273.615,Z 1648.306,A 0.000,B 0.000,C 90.000,E1 55.102} C_DIS
LIN {X 0.115,Y -260.991,Z 1648.288,A 0.000,B 0.000,C 90.000,E1 51.904} C_DIS
LIN {X 0.061,Y -249.003,Z 1648.271,A 0.000,B 0.000,C 90.000,E1 48.690} C_DIS
LIN {X -0.005,Y -237.812,Z 1648.252,A 0.000,B 0.000,C 90.000,E1 45.405} C_DIS
LIN {X -0.055,Y -227.298,Z 1648.234,A 0.000,B 0.000,C 90.000,E1 42.043} C_DIS
LIN {X -0.011,Y -217.630,Z 1648.214,A 0.000,B 0.000,C 90.000,E1 38.588} C_DIS
LIN {X -0.005,Y -209.829,Z 1648.197,A 0.000,B 0.000,C 90.000,E1 35.471} C_DIS
LIN {X 0.038,Y -202.740,Z 1648.179,A 0.000,B 0.000,C 90.000,E1 32.291} C_DIS
LIN {X 0.030,Y -196.379,Z 1648.162,A 0.000,B 0.000,C 90.000,E1 29.077} C_DIS
LIN {X -0.078,Y -190.625,Z 1648.143,A 0.000,B 0.000,C 90.000,E1 25.848} C_DIS
LIN {X 0.024,Y -185.583,Z 1648.125,A 0.000,B 0.000,C 90.000,E1 22.514} C_DIS
LIN {X -0.105,Y -181.236,Z 1648.107,A 0.000,B 0.000,C 90.000,E1 19.214} C_DIS
LIN {X 0.022,Y -176.810,Z 1648.083,A 0.000,B 0.000,C 90.000,E1 14.954} C_DIS
LIN {X -0.049,Y -173.245,Z 1648.059,A 0.000,B 0.000,C 90.000,E1 10.715} C_DIS
LIN {X -0.084,Y -170.064,Z 1648.031,A 0.000,B 0.000,C 90.000,E1 5.568} C_DIS
LIN {X -0.058,Y -167.764,Z 1647.993,A 0.000,B 0.000,C 90.000,E1 358.682} C_DIS
LIN {X 0.020,Y -168.871,Z 1647.930,A 0.000,B 0.000,C 90.000,E1 347.353} C_DIS
LIN {X -0.045,Y -171.784,Z 1647.901,A 0.000,B 0.000,C 90.000,E1 342.181} C_DIS
LIN {X 0.016,Y -174.721,Z 1647.882,A 0.000,B 0.000,C 90.000,E1 338.720} C_DIS
LIN {X 0.011,Y -178.507,Z 1647.863,A 0.000,B 0.000,C 90.000,E1 335.305} C_DIS
LIN {X 0.080,Y -183.151,Z 1647.844,A 0.000,B 0.000,C 90.000,E1 331.897} C_DIS
LIN {X -0.037,Y -188.601,Z 1647.825,A 0.000,B 0.000,C 90.000,E1 328.584} C_DIS
LIN {X 0.001,Y -193.233,Z 1647.812,A 0.000,B 0.000,C 90.000,E1 326.087} C_DIS
LIN {X -0.098,Y -200.344,Z 1647.793,A 0.000,B 0.000,C 90.000,E1 322.844} C_DIS
LIN {X 0.024,Y -207.319,Z 1647.778,A 0.000,B 0.000,C 90.000,E1 319.989} C_DIS
LIN {X -0.020,Y -215.243,Z 1647.762,A 0.000,B 0.000,C 90.000,E1 317.229} C_DIS
LIN {X -0.051,Y -224.079,Z 1647.747,A 0.000,B 0.000,C 90.000,E1 314.514} C_DIS
LIN {X 0.071,Y -235.369,Z 1647.730,A 0.000,B 0.000,C 90.000,E1 311.434} C_DIS
LIN {X 0.059,Y -244.812,Z 1647.718,A 0.000,B 0.000,C 90.000,E1 309.197} C_DIS
LIN {X -0.076,Y -255.337,Z 1647.706,A 0.000,B 0.000,C 90.000,E1 307.030} C_DIS
LIN {X -0.015,Y -267.051,Z 1647.694,A 0.000,B 0.000,C 90.000,E1 304.865} C_DIS
LIN {X -0.023,Y -282.058,Z 1647.680,A 0.000,B 0.000,C 90.000,E1 302.418} C_DIS
LIN {X 0.183,Y -300.913,Z 1647.665,A 0.000,B 0.000,C 90.000,E1 299.667} C_DIS
LIN {X 0.054,Y -315.937,Z 1647.654,A 0.000,B 0.000,C 90.000,E1 297.719} C_DIS
LIN {X 0.117,Y -328.278,Z 1647.645,A 0.000,B 0.000,C 90.000,E1 296.104} C_DIS
LIN {X -0.085,Y -340.447,Z 1647.636,A 0.000,B 0.000,C 90.000,E1 294.567} C_DIS
LIN {X -0.042,Y -354.920,Z 1647.626,A 0.000,B 0.000,C 90.000,E1 292.717} C_DIS
LIN {X -0.117,Y -366.914,Z 1647.618,A 0.000,B 0.000,C 90.000,E1 291.227} C_DIS
LIN {X 0.228,Y -376.164,Z 1647.611,A 0.000,B 0.000,C 90.000,E1 289.993} C_DIS
LIN {X 0.077,Y -382.623,Z 1647.606,A 0.000,B 0.000,C 90.000,E1 289.141} C_DIS
LIN {X -0.135,Y -388.570,Z 1647.602,A 0.000,B 0.000,C 90.000,E1 288.308} C_DIS
LIN {X -0.179,Y -393.897,Z 1647.597,A 0.000,B 0.000,C 90.000,E1 287.457} C_DIS
LIN {X 0.094,Y -398.355,Z 1647.592,A 0.000,B 0.000,C 90.000,E1 286.567} C_DIS
LIN {X -0.044,Y -400.824,Z 1647.589,A 0.000,B 0.000,C 90.000,E1 286.024} C_DIS
LIN {X 0.137,Y -401.922,Z 1647.587,A 0.000,B 0.000,C 90.000,E1 285.717} C_DIS
LIN {X -0.090,Y -403.769,Z 1647.584,A 0.000,B 0.000,C 90.000,E1 285.190} C_DIS
LIN {X 0.186,Y -405.331,Z 1647.581,A 0.000,B 0.000,C 90.000,E1 284.592} C_DIS
LIN {X -0.023,Y -406.475,Z 1647.578,A 0.000,B 0.000,C 90.000,E1 284.064} C_DIS
LIN {X -0.221,Y -407.207,Z 1647.575,A 0.000,B 0.000,C 90.000,E1 283.536} C_DIS
LIN {X 0.078,Y -407.474,Z 1647.572,A 0.000,B 0.000,C 90.000,E1 282.939} C_DIS
LIN {X -0.110,Y -407.281,Z 1647.569,A 0.000,B 0.000,C 90.000,E1 282.411} C_DIS
LIN {X 0.102,Y -406.613,Z 1647.566,A 0.000,B 0.000,C 90.000,E1 281.827} C_DIS
LIN {X -0.085,Y -405.358,Z 1647.563,A 0.000,B 0.000,C 90.000,E1 281.299} C_DIS
LIN {X 0.121,Y -403.493,Z 1647.560,A 0.000,B 0.000,C 90.000,E1 280.715} C_DIS
LIN {X -0.150,Y -401.072,Z 1647.557,A 0.000,B 0.000,C 90.000,E1 280.197} C_DIS
LIN {X 0.030,Y -397.925,Z 1647.553,A 0.000,B 0.000,C 90.000,E1 279.613} C_DIS
LIN {X 0.186,Y -394.200,Z 1647.550,A 0.000,B 0.000,C 90.000,E1 279.029} C_DIS
LIN {X -0.071,Y -387.786,Z 1647.546,A 0.000,B 0.000,C 90.000,E1 278.219} C_DIS
LIN {X 0.010,Y -380.830,Z 1647.541,A 0.000,B 0.000,C 90.000,E1 277.352} C_DIS
LIN {X 0.012,Y -375.554,Z 1647.538,A 0.000,B 0.000,C 90.000,E1 276.777} C_DIS
LIN {X 0.131,Y -369.800,Z 1647.535,A 0.000,B 0.000,C 90.000,E1 276.201} C_DIS
LIN {X 0.160,Y -363.758,Z 1647.532,A 0.000,B 0.000,C 90.000,E1 275.682} C_DIS
LIN {X 0.109,Y -357.508,Z 1647.529,A 0.000,B 0.000,C 90.000,E1 275.220} C_DIS
LIN {X -0.037,Y -351.025,Z 1647.527,A 0.000,B 0.000,C 90.000,E1 274.821} C_DIS
LIN {X 0.082,Y -341.464,Z 1647.524,A 0.000,B 0.000,C 90.000,E1 274.245} C_DIS
LIN {X 0.129,Y -331.769,Z 1647.521,A 0.000,B 0.000,C 90.000,E1 273.726} C_DIS
LIN {X 0.152,Y -322.027,Z 1647.518,A 0.000,B 0.000,C 90.000,E1 273.269} C_DIS
LIN {X 0.134,Y -311.925,Z 1647.516,A 0.000,B 0.000,C 90.000,E1 272.865} C_DIS
LIN {X 0.145,Y -301.708,Z 1647.514,A 0.000,B 0.000,C 90.000,E1 272.522} C_DIS
LIN {X 0.139,Y -290.659,Z 1647.513,A 0.000,B 0.000,C 90.000,E1 272.236} C_DIS
LIN {X -0.073,Y -283.048,Z 1647.512,A 0.000,B 0.000,C 90.000,E1 272.121} C_DIS
LIN {X 0.101,Y -272.977,Z 1647.511,A 0.000,B 0.000,C 90.000,E1 271.949} C_DIS
LIN {X -0.022,Y -237.422,Z 1647.510,A 0.000,B 0.000,C 90.000,E1 271.718} C_DIS
LIN {X -0.093,Y -213.712,Z 1647.509,A 0.000,B 0.000,C 90.000,E1 271.604} C_DIS
LIN {X 0.004,Y -188.586,Z 1647.508,A 0.000,B 0.000,C 90.000,E1 271.489} C_DIS
LIN {X -0.024,Y -181.355,Z 1647.508,A 0.000,B 0.000,C 90.000,E1 271.489} C_DIS
LIN {X 0.072,Y -181.550,Z 1647.503,A 0.000,B 0.000,C 90.000,E1 270.573} C_DIS
LIN {X 0.000,Y -181.299,Z 1647.494,A 0.000,B 0.000,C 90.000,E1 268.912} C_DIS
LIN {X 0.050,Y -180.907,Z 1647.475,A 0.000,B 0.000,C 90.000,E1 265.527} C_DIS
LIN {X -0.073,Y -180.767,Z 1647.471,A 0.000,B 0.000,C 90.000,E1 264.723} C_DIS
LIN {X -0.001,Y -178.862,Z 1647.442,A 0.000,B 0.000,C 90.000,E1 259.634} C_DIS
LIN {X 0.069,Y -175.905,Z 1647.414,A 0.000,B 0.000,C 90.000,E1 254.519} C_DIS
LIN {X 0.008,Y -174.588,Z 1647.405,A 0.000,B 0.000,C 90.000,E1 252.834} C_DIS
LIN {X 0.043,Y -171.571,Z 1647.381,A 0.000,B 0.000,C 90.000,E1 248.539} C_DIS
LIN {X 0.025,Y -167.793,Z 1647.357,A 0.000,B 0.000,C 90.000,E1 244.229} C_DIS
LIN {X 0.040,Y -166.510,Z 1647.347,A 0.000,B 0.000,C 90.000,E1 242.487} C_DIS
LIN {X 0.035,Y -163.218,Z 1647.328,A 0.000,B 0.000,C 90.000,E1 238.997} C_DIS
LIN {X -0.001,Y -161.184,Z 1647.313,A 0.000,B 0.000,C 90.000,E1 236.373} C_DIS
LIN {X -0.002,Y -157.196,Z 1647.289,A 0.000,B 0.000,C 90.000,E1 231.949} C_DIS
LIN {X 0.045,Y -155.925,Z 1647.279,A 0.000,B 0.000,C 90.000,E1 230.150} C_DIS
LIN {X -0.005,Y -152.176,Z 1647.254,A 0.000,B 0.000,C 90.000,E1 225.688} C_DIS
LIN {X 0.010,Y -150.424,Z 1647.239,A 0.000,B 0.000,C 90.000,E1 222.975} C_DIS
LIN {X -0.064,Y -147.151,Z 1647.214,A 0.000,B 0.000,C 90.000,E1 218.463} C_DIS
LIN {X 0.022,Y -145.166,Z 1647.193,A 0.000,B 0.000,C 90.000,E1 214.771} C_DIS
LIN {X -0.061,Y -142.318,Z 1647.163,A 0.000,B 0.000,C 90.000,E1 209.283} C_DIS
LIN {X 0.060,Y -141.708,Z 1647.152,A 0.000,B 0.000,C 90.000,E1 207.385} C_DIS
LIN {X -0.018,Y -139.470,Z 1647.116,A 0.000,B 0.000,C 90.000,E1 200.918} C_DIS
LIN {X 0.036,Y -139.202,Z 1647.106,A 0.000,B 0.000,C 90.000,E1 199.033} C_DIS
LIN {X -0.037,Y -138.329,Z 1647.054,A 0.000,B 0.000,C 90.000,E1 189.726} C_DIS
LIN {X -0.034,Y -139.441,Z 1647.007,A 0.000,B 0.000,C 90.000,E1 181.318} C_DIS
LIN {X 0.045,Y -140.976,Z 1646.976,A 0.000,B 0.000,C 90.000,E1 175.698} C_DIS
LIN {X -0.005,Y -142.731,Z 1646.956,A 0.000,B 0.000,C 90.000,E1 172.008} C_DIS
LIN {X -0.048,Y -145.118,Z 1646.930,A 0.000,B 0.000,C 90.000,E1 167.409} C_DIS
LIN {X -0.053,Y -147.743,Z 1646.910,A 0.000,B 0.000,C 90.000,E1 163.740} C_DIS
LIN {X 0.028,Y -150.409,Z 1646.889,A 0.000,B 0.000,C 90.000,E1 160.061} C_DIS
LIN {X 0.044,Y -153.846,Z 1646.869,A 0.000,B 0.000,C 90.000,E1 156.433} C_DIS
LIN {X -0.039,Y -157.256,Z 1646.849,A 0.000,B 0.000,C 90.000,E1 152.871} C_DIS
LIN {X 0.039,Y -161.431,Z 1646.829,A 0.000,B 0.000,C 90.000,E1 149.282} C_DIS
LIN {X 0.046,Y -165.633,Z 1646.810,A 0.000,B 0.000,C 90.000,E1 145.754} C_DIS
LIN {X 0.029,Y -170.563,Z 1646.790,A 0.000,B 0.000,C 90.000,E1 142.271} C_DIS
LIN {X -0.062,Y -175.441,Z 1646.771,A 0.000,B 0.000,C 90.000,E1 138.852} C_DIS
LIN {X 0.052,Y -181.065,Z 1646.752,A 0.000,B 0.000,C 90.000,E1 135.405} C_DIS
LIN {X -0.081,Y -186.502,Z 1646.734,A 0.000,B 0.000,C 90.000,E1 132.081} C_DIS
LIN {X -0.014,Y -191.122,Z 1646.720,A 0.000,B 0.000,C 90.000,E1 129.564} C_DIS
LIN {X -0.093,Y -196.919,Z 1646.702,A 0.000,B 0.000,C 90.000,E1 126.297} C_DIS
LIN {X 0.102,Y -200.181,Z 1646.693,A 0.000,B 0.000,C 90.000,E1 124.612} C_DIS
LIN {X -0.023,Y -206.813,Z 1646.672,A 0.000,B 0.000,C 90.000,E1 121.052} C_DIS
LIN {X -0.070,Y -327.321,Z 1646.672,A 0.000,B 0.000,C 90.000,E1 121.052} C_DIS
LIN {X 0.112,Y -328.552,Z 1646.672,A 0.000,B 0.000,C 90.000,E1 121.003} C_DIS
LIN {X 0.136,Y -333.452,Z 1646.671,A 0.000,B 0.000,C 90.000,E1 120.797} C_DIS
LIN {X 0.159,Y -336.041,Z 1646.670,A 0.000,B 0.000,C 90.000,E1 120.590} C_DIS
LIN {X 0.199,Y -339.841,Z 1646.668,A 0.000,B 0.000,C 90.000,E1 120.129} C_DIS
LIN {X -0.128,Y -341.644,Z 1646.666,A 0.000,B 0.000,C 90.000,E1 119.873} C_DIS
LIN {X 0.017,Y -356.773,Z 1646.647,A 0.000,B 0.000,C 90.000,E1 116.488} C_DIS
LIN {X -0.104,Y -370.688,Z 1646.632,A 0.000,B 0.000,C 90.000,E1 113.823} C_DIS
LIN {X 0.074,Y -384.404,Z 1646.619,A 0.000,B 0.000,C 90.000,E1 111.461} C_DIS
LIN {X -0.182,Y -399.483,Z 1646.607,A 0.000,B 0.000,C 90.000,E1 109.214} C_DIS
LIN {X -0.073,Y -416.029,Z 1646.594,A 0.000,B 0.000,C 90.000,E1 106.968} C_DIS
LIN {X 0.084,Y -434.158,Z 1646.582,A 0.000,B 0.000,C 90.000,E1 104.773} C_DIS
LIN {X -0.090,Y -453.761,Z 1646.571,A 0.000,B 0.000,C 90.000,E1 102.703} C_DIS
LIN {X -0.182,Y -474.035,Z 1646.560,A 0.000,B 0.000,C 90.000,E1 100.782} C_DIS
LIN {X -0.057,Y -499.939,Z 1646.548,A 0.000,B 0.000,C 90.000,E1 98.568} C_DIS
LIN {X 0.100,Y -501.840,Z 1646.546,A 0.000,B 0.000,C 90.000,E1 98.341} C_DIS
LIN {X 0.031,Y -503.518,Z 1646.545,A 0.000,B 0.000,C 90.000,E1 98.106} C_DIS
LIN {X -0.043,Y -504.771,Z 1646.544,A 0.000,B 0.000,C 90.000,E1 97.871} C_DIS
LIN {X 0.263,Y -506.295,Z 1646.541,A 0.000,B 0.000,C 90.000,E1 97.352} C_DIS
LIN {X 0.075,Y -506.739,Z 1646.538,A 0.000,B 0.000,C 90.000,E1 96.891} C_DIS
LIN {X -0.105,Y -506.175,Z 1646.536,A 0.000,B 0.000,C 90.000,E1 96.429} C_DIS
LIN {X 0.219,Y -504.511,Z 1646.533,A 0.000,B 0.000,C 90.000,E1 95.910} C_DIS
LIN {X 0.103,Y -503.171,Z 1646.532,A 0.000,B 0.000,C 90.000,E1 95.682} C_DIS
LIN {X -0.159,Y -491.213,Z 1646.522,A 0.000,B 0.000,C 90.000,E1 94.012} C_DIS
LIN {X -0.229,Y -479.114,Z 1646.513,A 0.000,B 0.000,C 90.000,E1 92.293} C_DIS
LIN {X 0.139,Y -468.539,Z 1646.504,A 0.000,B 0.000,C 90.000,E1 90.745} C_DIS
LIN {X -0.155,Y -457.674,Z 1646.496,A 0.000,B 0.000,C 90.000,E1 89.255} C_DIS
LIN {X 0.082,Y -448.387,Z 1646.489,A 0.000,B 0.000,C 90.000,E1 87.936} C_DIS
LIN {X -0.087,Y -436.778,Z 1646.480,A 0.000,B 0.000,C 90.000,E1 86.388} C_DIS
LIN {X -0.142,Y -421.109,Z 1646.468,A 0.000,B 0.000,C 90.000,E1 84.261} C_DIS
LIN {X 0.189,Y -400.234,Z 1646.451,A 0.000,B 0.000,C 90.000,E1 81.197} C_DIS
LIN {X -0.068,Y -382.588,Z 1646.436,A 0.000,B 0.000,C 90.000,E1 78.409} C_DIS
LIN {X -0.130,Y -367.478,Z 1646.421,A 0.000,B 0.000,C 90.000,E1 75.811} C_DIS
LIN {X -0.144,Y -352.960,Z 1646.406,A 0.000,B 0.000,C 90.000,E1 73.142} C_DIS
LIN {X 0.081,Y -336.170,Z 1646.388,A 0.000,B 0.000,C 90.000,E1 69.752} C_DIS
LIN {X 0.080,Y -320.323,Z 1646.368,A 0.000,B 0.000,C 90.000,E1 66.305} C_DIS
LIN {X -0.026,Y -308.142,Z 1646.352,A 0.000,B 0.000,C 90.000,E1 63.435} C_DIS
LIN {X 0.033,Y -300.091,Z 1646.342,A 0.000,B 0.000,C 90.000,E1 61.463} C_DIS
LIN {X 0.104,Y -291.916,Z 1646.330,A 0.000,B 0.000,C 90.000,E1 59.459} C_DIS
LIN {X 0.026,Y -283.487,Z 1646.319,A 0.000,B 0.000,C 90.000,E1 57.454} C_DIS
LIN {X 0.094,Y -274.874,Z 1646.308,A 0.000,B 0.000,C 90.000,E1 55.388} C_DIS
LIN {X -0.018,Y -262.203,Z 1646.290,A 0.000,B 0.000,C 90.000,E1 52.271} C_DIS
LIN {X -0.029,Y -250.110,Z 1646.272,A 0.000,B 0.000,C 90.000,E1 49.057} C_DIS
LIN {X 0.112,Y -238.789,Z 1646.254,A 0.000,B 0.000,C 90.000,E1 45.729} C_DIS
LIN {X 0.089,Y -228.200,Z 1646.235,A 0.000,B 0.000,C 90.000,E1 42.366} C_DIS
LIN {X -0.088,Y -219.460,Z 1646.219,A 0.000,B 0.000,C 90.000,E1 39.358} C_DIS
LIN {X 0.053,Y -211.456,Z 1646.201,A 0.000,B 0.000,C 90.000,E1 36.217} C_DIS
LIN {X -0.043,Y -204.205,Z 1646.184,A 0.000,B 0.000,C 90.000,E1 33.086} C_DIS
LIN {X -0.015,Y -197.719,Z 1646.166,A 0.000,B 0.000,C 90.000,E1 29.873} C_DIS
LIN {X 0.001,Y -191.874,Z 1646.148,A 0.000,B 0.000,C 90.000,E1 26.616} C_DIS
LIN {X -0.036,Y -186.701,Z 1646.130,A 0.000,B 0.000,C 90.000,E1 23.334} C_DIS
LIN {X -0.006,Y -182.197,Z 1646.111,A 0.000,B 0.000,C 90.000,E1 19.993} C_DIS
LIN {X -0.026,Y -177.640,Z 1646.088,A 0.000,B 0.000,C 90.000,E1 15.788} C_DIS
LIN {X -0.028,Y -173.917,Z 1646.064,A 0.000,B 0.000,C 90.000,E1 11.535} C_DIS
LIN {X 0.006,Y -170.558,Z 1646.035,A 0.000,B 0.000,C 90.000,E1 6.372} C_DIS
LIN {X -0.030,Y -167.996,Z 1645.997,A 0.000,B 0.000,C 90.000,E1 359.542} C_DIS
LIN {X 0.027,Y -168.959,Z 1645.930,A 0.000,B 0.000,C 90.000,E1 347.353} C_DIS
LIN {X -0.034,Y -171.907,Z 1645.901,A 0.000,B 0.000,C 90.000,E1 342.181} C_DIS
LIN {X 0.030,Y -174.844,Z 1645.882,A 0.000,B 0.000,C 90.000,E1 338.720} C_DIS
LIN {X 0.028,Y -178.628,Z 1645.863,A 0.000,B 0.000,C 90.000,E1 335.305} C_DIS
LIN {X 0.100,Y -183.300,Z 1645.844,A 0.000,B 0.000,C 90.000,E1 331.897} C_DIS
LIN {X -0.012,Y -188.768,Z 1645.825,A 0.000,B 0.000,C 90.000,E1 328.584} C_DIS
LIN {X 0.043,Y -195.104,Z 1645.807,A 0.000,B 0.000,C 90.000,E1 325.261} C_DIS
LIN {X -0.050,Y -202.416,Z 1645.789,A 0.000,B 0.000,C 90.000,E1 322.029} C_DIS
LIN {X -0.029,Y -209.635,Z 1645.773,A 0.000,B 0.000,C 90.000,E1 319.218} C_DIS
LIN {X -0.022,Y -217.809,Z 1645.758,A 0.000,B 0.000,C 90.000,E1 316.458} C_DIS
LIN {X 0.005,Y -226.912,Z 1645.743,A 0.000,B 0.000,C 90.000,E1 313.743} C_DIS
LIN {X 0.051,Y -238.491,Z 1645.726,A 0.000,B 0.000,C 90.000,E1 310.701} C_DIS
LIN {X 0.105,Y -248.241,Z 1645.714,A 0.000,B 0.000,C 90.000,E1 308.463} C_DIS
LIN {X 0.037,Y -259.123,Z 1645.702,A 0.000,B 0.000,C 90.000,E1 306.297} C_DIS
LIN {X -0.071,Y -273.322,Z 1645.688,A 0.000,B 0.000,C 90.000,E1 303.833} C_DIS
LIN {X -0.046,Y -286.627,Z 1645.676,A 0.000,B 0.000,C 90.000,E1 301.750} C_DIS
LIN {X -0.106,Y -308.398,Z 1645.660,A 0.000,B 0.000,C 90.000,E1 298.743} C_DIS
LIN {X 0.105,Y -320.900,Z 1645.651,A 0.000,B 0.000,C 90.000,E1 297.078} C_DIS
LIN {X -0.050,Y -333.182,Z 1645.642,A 0.000,B 0.000,C 90.000,E1 295.515} C_DIS
LIN {X -0.010,Y -347.683,Z 1645.631,A 0.000,B 0.000,C 90.000,E1 293.643} C_DIS
LIN {X -0.150,Y -362.130,Z 1645.621,A 0.000,B 0.000,C 90.000,E1 291.844} C_DIS
LIN {X -0.131,Y -373.895,Z 1645.613,A 0.000,B 0.000,C 90.000,E1 290.355} C_DIS
LIN {X 0.056,Y -380.484,Z 1645.608,A 0.000,B 0.000,C 90.000,E1 289.450} C_DIS
LIN {X -0.058,Y -386.645,Z 1645.603,A 0.000,B 0.000,C 90.000,E1 288.598} C_DIS
LIN {X -0.115,Y -392.177,Z 1645.599,A 0.000,B 0.000,C 90.000,E1 287.747} C_DIS
LIN {X 0.132,Y -397.032,Z 1645.594,A 0.000,B 0.000,C 90.000,E1 286.858} C_DIS
LIN {X -0.015,Y -399.721,Z 1645.591,A 0.000,B 0.000,C 90.000,E1 286.315} C_DIS
LIN {X 0.129,Y -401.986,Z 1645.588,A 0.000,B 0.000,C 90.000,E1 285.733} C_DIS
LIN {X 0.011,Y -403.911,Z 1645.584,A 0.000,B 0.000,C 90.000,E1 285.190} C_DIS
LIN {X -0.105,Y -405.469,Z 1645.581,A 0.000,B 0.000,C 90.000,E1 284.647} C_DIS
LIN {X 0.080,Y -406.646,Z 1645.578,A 0.000,B 0.000,C 90.000,E1 284.064} C_DIS
LIN {X -0.117,Y -407.373,Z 1645.575,A 0.000,B 0.000,C 90.000,E1 283.536} C_DIS
LIN {X 0.183,Y -407.713,Z 1645.572,A 0.000,B 0.000,C 90.000,E1 282.939} C_DIS
LIN {X -0.004,Y -407.516,Z 1645.569,A 0.000,B 0.000,C 90.000,E1 282.411} C_DIS
LIN {X 0.209,Y -406.871,Z 1645.566,A 0.000,B 0.000,C 90.000,E1 281.827} C_DIS
LIN {X 0.023,Y -405.654,Z 1645.563,A 0.000,B 0.000,C 90.000,E1 281.299} C_DIS
LIN {X 0.154,Y -403.815,Z 1645.560,A 0.000,B 0.000,C 90.000,E1 280.725} C_DIS
LIN {X -0.040,Y -401.388,Z 1645.557,A 0.000,B 0.000,C 90.000,E1 280.197} C_DIS
LIN {X 0.140,Y -398.248,Z 1645.553,A 0.000,B 0.000,C 90.000,E1 279.613} C_DIS
LIN {X -0.152,Y -394.516,Z 1645.550,A 0.000,B 0.000,C 90.000,E1 279.095} C_DIS
LIN {X 0.043,Y -388.069,Z 1645.546,A 0.000,B 0.000,C 90.000,E1 278.219} C_DIS
LIN {X 0.123,Y -381.092,Z 1645.541,A 0.000,B 0.000,C 90.000,E1 277.352} C_DIS
LIN {X 0.126,Y -375.800,Z 1645.538,A 0.000,B 0.000,C 90.000,E1 276.777} C_DIS
LIN {X -0.113,Y -370.054,Z 1645.535,A 0.000,B 0.000,C 90.000,E1 276.258} C_DIS
LIN {X -0.078,Y -364.000,Z 1645.532,A 0.000,B 0.000,C 90.000,E1 275.739} C_DIS
LIN {X -0.136,Y -357.704,Z 1645.529,A 0.000,B 0.000,C 90.000,E1 275.277} C_DIS
LIN {X 0.095,Y -351.363,Z 1645.527,A 0.000,B 0.000,C 90.000,E1 274.821} C_DIS
LIN {X -0.168,Y -341.673,Z 1645.524,A 0.000,B 0.000,C 90.000,E1 274.302} C_DIS
LIN {X -0.137,Y -331.930,Z 1645.521,A 0.000,B 0.000,C 90.000,E1 273.784} C_DIS
LIN {X -0.095,Y -322.138,Z 1645.518,A 0.000,B 0.000,C 90.000,E1 273.326} C_DIS
LIN {X -0.055,Y -312.239,Z 1645.516,A 0.000,B 0.000,C 90.000,E1 272.922} C_DIS
LIN {X -0.026,Y -302.110,Z 1645.514,A 0.000,B 0.000,C 90.000,E1 272.579} C_DIS
LIN {X -0.005,Y -291.353,Z 1645.513,A 0.000,B 0.000,C 90.000,E1 272.293} C_DIS
LIN {X 0.045,Y -283.468,Z 1645.512,A 0.000,B 0.000,C 90.000,E1 272.121} C_DIS
LIN {X -0.060,Y -273.555,Z 1645.511,A 0.000,B 0.000,C 90.000,E1 272.007} C_DIS
LIN {X 0.073,Y -239.079,Z 1645.510,A 0.000,B 0.000,C 90.000,E1 271.718} C_DIS
LIN {X -0.018,Y -217.715,Z 1645.509,A 0.000,B 0.000,C 90.000,E1 271.604} C_DIS
LIN {X 0.063,Y -189.348,Z 1645.508,A 0.000,B 0.000,C 90.000,E1 271.489} C_DIS
LIN {X 0.029,Y -181.351,Z 1645.508,A 0.000,B 0.000,C 90.000,E1 271.489} C_DIS
LIN {X -0.071,Y -181.547,Z 1645.503,A 0.000,B 0.000,C 90.000,E1 270.630} C_DIS
LIN {X 0.039,Y -181.302,Z 1645.494,A 0.000,B 0.000,C 90.000,E1 268.912} C_DIS
LIN {X 0.088,Y -180.908,Z 1645.475,A 0.000,B 0.000,C 90.000,E1 265.527} C_DIS
LIN {X -0.034,Y -180.772,Z 1645.471,A 0.000,B 0.000,C 90.000,E1 264.723} C_DIS
LIN {X 0.037,Y -178.868,Z 1645.443,A 0.000,B 0.000,C 90.000,E1 259.634} C_DIS
LIN {X -0.062,Y -175.911,Z 1645.414,A 0.000,B 0.000,C 90.000,E1 254.574} C_DIS
LIN {X -0.006,Y -174.598,Z 1645.405,A 0.000,B 0.000,C 90.000,E1 252.851} C_DIS
LIN {X -0.079,Y -171.580,Z 1645.381,A 0.000,B 0.000,C 90.000,E1 248.592} C_DIS
LIN {X -0.089,Y -167.803,Z 1645.357,A 0.000,B 0.000,C 90.000,E1 244.280} C_DIS
LIN {X 0.076,Y -166.521,Z 1645.347,A 0.000,B 0.000,C 90.000,E1 242.487} C_DIS
LIN {X 0.064,Y -162.522,Z 1645.323,A 0.000,B 0.000,C 90.000,E1 238.122} C_DIS
LIN {X 0.036,Y -161.196,Z 1645.313,A 0.000,B 0.000,C 90.000,E1 236.373} C_DIS
LIN {X -0.063,Y -157.206,Z 1645.289,A 0.000,B 0.000,C 90.000,E1 231.984} C_DIS
LIN {X -0.039,Y -155.934,Z 1645.279,A 0.000,B 0.000,C 90.000,E1 230.194} C_DIS
LIN {X -0.080,Y -152.186,Z 1645.254,A 0.000,B 0.000,C 90.000,E1 225.729} C_DIS
LIN {X -0.058,Y -150.432,Z 1645.239,A 0.000,B 0.000,C 90.000,E1 223.014} C_DIS
LIN {X -0.030,Y -147.159,Z 1645.214,A 0.000,B 0.000,C 90.000,E1 218.463} C_DIS
LIN {X -0.063,Y -145.175,Z 1645.193,A 0.000,B 0.000,C 90.000,E1 214.818} C_DIS
LIN {X -0.027,Y -142.324,Z 1645.163,A 0.000,B 0.000,C 90.000,E1 209.283} C_DIS
LIN {X -0.033,Y -141.713,Z 1645.152,A 0.000,B 0.000,C 90.000,E1 207.436} C_DIS
LIN {X 0.015,Y -139.473,Z 1645.116,A 0.000,B 0.000,C 90.000,E1 200.918} C_DIS
LIN {X -0.062,Y -139.205,Z 1645.106,A 0.000,B 0.000,C 90.000,E1 199.087} C_DIS
LIN {X -0.004,Y -138.330,Z 1645.054,A 0.000,B 0.000,C 90.000,E1 189.726} C_DIS
LIN {X -0.001,Y -139.438,Z 1645.007,A 0.000,B 0.000,C 90.000,E1 181.318} C_DIS
LIN {X -0.062,Y -140.970,Z 1644.976,A 0.000,B 0.000,C 90.000,E1 175.755} C_DIS
LIN {X 0.029,Y -142.725,Z 1644.956,A 0.000,B 0.000,C 90.000,E1 172.008} C_DIS
LIN {X -0.013,Y -145.110,Z 1644.930,A 0.000,B 0.000,C 90.000,E1 167.409} C_DIS
LIN {X -0.018,Y -147.733,Z 1644.910,A 0.000,B 0.000,C 90.000,E1 163.740} C_DIS
LIN {X 0.063,Y -150.397,Z 1644.889,A 0.000,B 0.000,C 90.000,E1 160.061} C_DIS
LIN {X -0.062,Y -153.832,Z 1644.869,A 0.000,B 0.000,C 90.000,E1 156.485} C_DIS
LIN {X -0.003,Y -157.243,Z 1644.849,A 0.000,B 0.000,C 90.000,E1 152.871} C_DIS
LIN {X -0.063,Y -161.414,Z 1644.829,A 0.000,B 0.000,C 90.000,E1 149.331} C_DIS
LIN {X -0.053,Y -165.616,Z 1644.810,A 0.000,B 0.000,C 90.000,E1 145.801} C_DIS
LIN {X 0.067,Y -170.544,Z 1644.791,A 0.000,B 0.000,C 90.000,E1 142.271} C_DIS
LIN {X -0.025,Y -175.422,Z 1644.771,A 0.000,B 0.000,C 90.000,E1 138.852} C_DIS
LIN {X 0.092,Y -181.046,Z 1644.752,A 0.000,B 0.000,C 90.000,E1 135.405} C_DIS
LIN {X -0.041,Y -186.480,Z 1644.734,A 0.000,B 0.000,C 90.000,E1 132.081} C_DIS
LIN {X 0.026,Y -191.103,Z 1644.720,A 0.000,B 0.000,C 90.000,E1 129.564} C_DIS
LIN {X -0.053,Y -196.896,Z 1644.702,A 0.000,B 0.000,C 90.000,E1 126.297} C_DIS
LIN {X -0.022,Y -200.156,Z 1644.693,A 0.000,B 0.000,C 90.000,E1 124.659} C_DIS
LIN {X 0.019,Y -206.730,Z 1644.673,A 0.000,B 0.000,C 90.000,E1 121.082} C_DIS
LIN {X -0.006,Y -327.076,Z 1644.673,A 0.000,B 0.000,C 90.000,E1 121.082} C_DIS
LIN {X -0.118,Y -333.352,Z 1644.671,A 0.000,B 0.000,C 90.000,E1 120.875} C_DIS
LIN {X 0.056,Y -336.158,Z 1644.670,A 0.000,B 0.000,C 90.000,E1 120.620} C_DIS
LIN {X 0.205,Y -339.908,Z 1644.668,A 0.000,B 0.000,C 90.000,E1 120.129} C_DIS
LIN {X -0.120,Y -341.651,Z 1644.666,A 0.000,B 0.000,C 90.000,E1 119.873} C_DIS
LIN {X 0.024,Y -356.747,Z 1644.647,A 0.000,B 0.000,C 90.000,E1 116.488} C_DIS
LIN {X -0.098,Y -370.660,Z 1644.632,A 0.000,B 0.000,C 90.000,E1 113.823} C_DIS
LIN {X 0.079,Y -384.375,Z 1644.619,A 0.000,B 0.000,C 90.000,E1 111.461} C_DIS
LIN {X -0.178,Y -399.452,Z 1644.607,A 0.000,B 0.000,C 90.000,E1 109.214} C_DIS
LIN {X -0.068,Y -415.998,Z 1644.594,A 0.000,B 0.000,C 90.000,E1 106.968} C_DIS
LIN {X 0.088,Y -434.127,Z 1644.582,A 0.000,B 0.000,C 90.000,E1 104.773} C_DIS
LIN {X -0.088,Y -453.729,Z 1644.571,A 0.000,B 0.000,C 90.000,E1 102.703} C_DIS
LIN {X -0.180,Y -474.003,Z 1644.560,A 0.000,B 0.000,C 90.000,E1 100.782} C_DIS
LIN {X -0.057,Y -499.882,Z 1644.548,A 0.000,B 0.000,C 90.000,E1 98.568} C_DIS
LIN {X 0.101,Y -501.753,Z 1644.546,A 0.000,B 0.000,C 90.000,E1 98.341} C_DIS
LIN {X 0.030,Y -503.408,Z 1644.545,A 0.000,B 0.000,C 90.000,E1 98.106} C_DIS
LIN {X -0.042,Y -504.643,Z 1644.544,A 0.000,B 0.000,C 90.000,E1 97.871} C_DIS
LIN {X 0.262,Y -506.137,Z 1644.541,A 0.000,B 0.000,C 90.000,E1 97.352} C_DIS
LIN {X 0.074,Y -506.555,Z 1644.538,A 0.000,B 0.000,C 90.000,E1 96.891} C_DIS
LIN {X -0.107,Y -505.966,Z 1644.536,A 0.000,B 0.000,C 90.000,E1 96.429} C_DIS
LIN {X 0.216,Y -504.272,Z 1644.533,A 0.000,B 0.000,C 90.000,E1 95.910} C_DIS
LIN {X 0.099,Y -502.912,Z 1644.532,A 0.000,B 0.000,C 90.000,E1 95.682} C_DIS
LIN {X 0.177,Y -489.280,Z 1644.521,A 0.000,B 0.000,C 90.000,E1 93.726} C_DIS
LIN {X 0.071,Y -477.166,Z 1644.511,A 0.000,B 0.000,C 90.000,E1 92.007} C_DIS
LIN {X -0.069,Y -466.544,Z 1644.503,A 0.000,B 0.000,C 90.000,E1 90.516} C_DIS
LIN {X 0.066,Y -455.636,Z 1644.494,A 0.000,B 0.000,C 90.000,E1 88.969} C_DIS
LIN {X -0.184,Y -446.275,Z 1644.487,A 0.000,B 0.000,C 90.000,E1 87.707} C_DIS
LIN {X 0.050,Y -434.571,Z 1644.478,A 0.000,B 0.000,C 90.000,E1 86.102} C_DIS
LIN {X -0.171,Y -420.851,Z 1644.468,A 0.000,B 0.000,C 90.000,E1 84.261} C_DIS
LIN {X 0.152,Y -399.944,Z 1644.451,A 0.000,B 0.000,C 90.000,E1 81.197} C_DIS
LIN {X -0.111,Y -382.289,Z 1644.436,A 0.000,B 0.000,C 90.000,E1 78.409} C_DIS
LIN {X 0.177,Y -367.206,Z 1644.421,A 0.000,B 0.000,C 90.000,E1 75.755} C_DIS
LIN {X 0.138,Y -352.682,Z 1644.406,A 0.000,B 0.000,C 90.000,E1 73.087} C_DIS
LIN {X 0.021,Y -335.919,Z 1644.388,A 0.000,B 0.000,C 90.000,E1 69.752} C_DIS
LIN {X 0.013,Y -320.046,Z 1644.368,A 0.000,B 0.000,C 90.000,E1 66.305} C_DIS
LIN {X -0.097,Y -307.899,Z 1644.352,A 0.000,B 0.000,C 90.000,E1 63.435} C_DIS
LIN {X -0.022,Y -298.500,Z 1644.340,A 0.000,B 0.000,C 90.000,E1 61.129} C_DIS
LIN {X 0.023,Y -290.300,Z 1644.328,A 0.000,B 0.000,C 90.000,E1 59.125} C_DIS
LIN {X -0.052,Y -283.296,Z 1644.319,A 0.000,B 0.000,C 90.000,E1 57.454} C_DIS
LIN {X 0.015,Y -274.710,Z 1644.308,A 0.000,B 0.000,C 90.000,E1 55.388} C_DIS
LIN {X -0.098,Y -262.032,Z 1644.290,A 0.000,B 0.000,C 90.000,E1 52.271} C_DIS
LIN {X 0.079,Y -249.916,Z 1644.272,A 0.000,B 0.000,C 90.000,E1 49.013} C_DIS
LIN {X 0.029,Y -238.554,Z 1644.254,A 0.000,B 0.000,C 90.000,E1 45.729} C_DIS
LIN {X 0.003,Y -227.950,Z 1644.235,A 0.000,B 0.000,C 90.000,E1 42.366} C_DIS
LIN {X -0.038,Y -219.202,Z 1644.218,A 0.000,B 0.000,C 90.000,E1 39.322} C_DIS
LIN {X -0.039,Y -211.206,Z 1644.201,A 0.000,B 0.000,C 90.000,E1 36.217} C_DIS
LIN {X 0.034,Y -203.987,Z 1644.184,A 0.000,B 0.000,C 90.000,E1 33.038} C_DIS
LIN {X -0.112,Y -197.536,Z 1644.166,A 0.000,B 0.000,C 90.000,E1 29.873} C_DIS
LIN {X -0.098,Y -191.743,Z 1644.148,A 0.000,B 0.000,C 90.000,E1 26.616} C_DIS
LIN {X 0.036,Y -186.613,Z 1644.129,A 0.000,B 0.000,C 90.000,E1 23.281} C_DIS
LIN {X 0.067,Y -182.174,Z 1644.111,A 0.000,B 0.000,C 90.000,E1 19.939} C_DIS
LIN {X 0.049,Y -177.654,Z 1644.088,A 0.000,B 0.000,C 90.000,E1 15.733} C_DIS
LIN {X 0.048,Y -173.945,Z 1644.064,A 0.000,B 0.000,C 90.000,E1 11.478} C_DIS
LIN {X 0.085,Y -170.613,Z 1644.035,A 0.000,B 0.000,C 90.000,E1 6.315} C_DIS
LIN {X -0.030,Y -168.098,Z 1643.997,A 0.000,B 0.000,C 90.000,E1 359.542} C_DIS
LIN {X 0.010,Y -168.711,Z 1643.935,A 0.000,B 0.000,C 90.000,E1 348.229} C_DIS
LIN {X 0.064,Y -171.428,Z 1643.906,A 0.000,B 0.000,C 90.000,E1 343.015} C_DIS
LIN {X 0.044,Y -174.966,Z 1643.882,A 0.000,B 0.000,C 90.000,E1 338.720} C_DIS
LIN {X 0.046,Y -178.749,Z 1643.863,A 0.000,B 0.000,C 90.000,E1 335.305} C_DIS
LIN {X -0.039,Y -183.449,Z 1643.844,A 0.000,B 0.000,C 90.000,E1 331.948} C_DIS
LIN {X 0.014,Y -188.943,Z 1643.825,A 0.000,B 0.000,C 90.000,E1 328.584} C_DIS
LIN {X 0.075,Y -195.292,Z 1643.807,A 0.000,B 0.000,C 90.000,E1 325.261} C_DIS
LIN {X -0.012,Y -202.584,Z 1643.789,A 0.000,B 0.000,C 90.000,E1 322.029} C_DIS
LIN {X 0.013,Y -209.782,Z 1643.773,A 0.000,B 0.000,C 90.000,E1 319.218} C_DIS
LIN {X 0.026,Y -217.943,Z 1643.758,A 0.000,B 0.000,C 90.000,E1 316.458} C_DIS
LIN {X -0.020,Y -228.393,Z 1643.741,A 0.000,B 0.000,C 90.000,E1 313.380} C_DIS
LIN {X 0.110,Y -238.552,Z 1643.726,A 0.000,B 0.000,C 90.000,E1 310.701} C_DIS
LIN {X -0.028,Y -248.295,Z 1643.714,A 0.000,B 0.000,C 90.000,E1 308.508} C_DIS
LIN {X 0.102,Y -259.156,Z 1643.702,A 0.000,B 0.000,C 90.000,E1 306.297} C_DIS
LIN {X -0.002,Y -273.325,Z 1643.688,A 0.000,B 0.000,C 90.000,E1 303.833} C_DIS
LIN {X -0.004,Y -288.955,Z 1643.675,A 0.000,B 0.000,C 90.000,E1 301.416} C_DIS
LIN {X -0.003,Y -310.940,Z 1643.658,A 0.000,B 0.000,C 90.000,E1 298.409} C_DIS
LIN {X -0.027,Y -323.359,Z 1643.649,A 0.000,B 0.000,C 90.000,E1 296.796} C_DIS
LIN {X -0.006,Y -335.605,Z 1643.640,A 0.000,B 0.000,C 90.000,E1 295.207} C_DIS
LIN {X 0.087,Y -350.087,Z 1643.630,A 0.000,B 0.000,C 90.000,E1 293.334} C_DIS
LIN {X -0.003,Y -364.497,Z 1643.620,A 0.000,B 0.000,C 90.000,E1 291.535} C_DIS
LIN {X -0.036,Y -373.852,Z 1643.613,A 0.000,B 0.000,C 90.000,E1 290.355} C_DIS
LIN {X -0.218,Y -382.583,Z 1643.607,A 0.000,B 0.000,C 90.000,E1 289.214} C_DIS
LIN {X 0.059,Y -388.548,Z 1643.602,A 0.000,B 0.000,C 90.000,E1 288.308} C_DIS
LIN {X 0.018,Y -393.929,Z 1643.597,A 0.000,B 0.000,C 90.000,E1 287.457} C_DIS
LIN {X -0.088,Y -398.459,Z 1643.592,A 0.000,B 0.000,C 90.000,E1 286.622} C_DIS
LIN {X -0.156,Y -402.070,Z 1643.588,A 0.000,B 0.000,C 90.000,E1 285.788} C_DIS
LIN {X 0.113,Y -404.022,Z 1643.584,A 0.000,B 0.000,C 90.000,E1 285.190} C_DIS
LIN {X -0.002,Y -405.629,Z 1643.581,A 0.000,B 0.000,C 90.000,E1 284.647} C_DIS
LIN {X 0.185,Y -406.820,Z 1643.578,A 0.000,B 0.000,C 90.000,E1 284.064} C_DIS
LIN {X -0.012,Y -407.608,Z 1643.575,A 0.000,B 0.000,C 90.000,E1 283.536} C_DIS
LIN {X -0.199,Y -407.938,Z 1643.572,A 0.000,B 0.000,C 90.000,E1 283.008} C_DIS
LIN {X 0.104,Y -407.798,Z 1643.569,A 0.000,B 0.000,C 90.000,E1 282.411} C_DIS
LIN {X -0.080,Y -407.130,Z 1643.566,A 0.000,B 0.000,C 90.000,E1 281.883} C_DIS
LIN {X 0.134,Y -405.959,Z 1643.563,A 0.000,B 0.000,C 90.000,E1 281.299} C_DIS
LIN {X -0.130,Y -404.184,Z 1643.560,A 0.000,B 0.000,C 90.000,E1 280.782} C_DIS
LIN {X -0.028,Y -403.055,Z 1643.558,A 0.000,B 0.000,C 90.000,E1 280.489} C_DIS
LIN {X 0.164,Y -400.272,Z 1643.555,A 0.000,B 0.000,C 90.000,E1 279.905} C_DIS
LIN {X -0.055,Y -396.789,Z 1643.552,A 0.000,B 0.000,C 90.000,E1 279.378} C_DIS
LIN {X 0.103,Y -390.655,Z 1643.547,A 0.000,B 0.000,C 90.000,E1 278.511} C_DIS
LIN {X -0.179,Y -383.809,Z 1643.543,A 0.000,B 0.000,C 90.000,E1 277.701} C_DIS
LIN {X -0.157,Y -378.832,Z 1643.539,A 0.000,B 0.000,C 90.000,E1 277.125} C_DIS
LIN {X -0.083,Y -373.298,Z 1643.536,A 0.000,B 0.000,C 90.000,E1 276.549} C_DIS
LIN {X -0.131,Y -367.394,Z 1643.533,A 0.000,B 0.000,C 90.000,E1 276.024} C_DIS
LIN {X 0.007,Y -361.300,Z 1643.531,A 0.000,B 0.000,C 90.000,E1 275.511} C_DIS
LIN {X 0.108,Y -354.915,Z 1643.528,A 0.000,B 0.000,C 90.000,E1 275.049} C_DIS
LIN {X 0.006,Y -345.257,Z 1643.525,A 0.000,B 0.000,C 90.000,E1 274.473} C_DIS
LIN {X -0.004,Y -335.670,Z 1643.522,A 0.000,B 0.000,C 90.000,E1 273.955} C_DIS
LIN {X -0.142,Y -325.723,Z 1643.519,A 0.000,B 0.000,C 90.000,E1 273.498} C_DIS
LIN {X 0.120,Y -315.875,Z 1643.517,A 0.000,B 0.000,C 90.000,E1 273.037} C_DIS
LIN {X 0.013,Y -305.670,Z 1643.515,A 0.000,B 0.000,C 90.000,E1 272.694} C_DIS
LIN {X -0.062,Y -295.019,Z 1643.513,A 0.000,B 0.000,C 90.000,E1 272.407} C_DIS
LIN {X 0.117,Y -283.587,Z 1643.512,A 0.000,B 0.000,C 90.000,E1 272.121} C_DIS
LIN {X 0.004,Y -273.111,Z 1643.511,A 0.000,B 0.000,C 90.000,E1 272.007} C_DIS
LIN {X 0.011,Y -243.775,Z 1643.510,A 0.000,B 0.000,C 90.000,E1 271.776} C_DIS
LIN {X 0.086,Y -220.841,Z 1643.509,A 0.000,B 0.000,C 90.000,E1 271.604} C_DIS
LIN {X -0.065,Y -190.333,Z 1643.509,A 0.000,B 0.000,C 90.000,E1 271.547} C_DIS
LIN {X -0.088,Y -181.348,Z 1643.508,A 0.000,B 0.000,C 90.000,E1 271.547} C_DIS
LIN {X -0.059,Y -181.558,Z 1643.500,A 0.000,B 0.000,C 90.000,E1 270.000} C_DIS
LIN {X 0.077,Y -180.901,Z 1643.474,A 0.000,B 0.000,C 90.000,E1 265.241} C_DIS
LIN {X 0.027,Y -180.228,Z 1643.464,A 0.000,B 0.000,C 90.000,E1 263.571} C_DIS
LIN {X -0.020,Y -179.042,Z 1643.446,A 0.000,B 0.000,C 90.000,E1 260.208} C_DIS
LIN {X 0.043,Y -178.710,Z 1643.441,A 0.000,B 0.000,C 90.000,E1 259.342} C_DIS
LIN {X -0.065,Y -175.759,Z 1643.413,A 0.000,B 0.000,C 90.000,E1 254.283} C_DIS
LIN {X -0.014,Y -171.943,Z 1643.384,A 0.000,B 0.000,C 90.000,E1 249.135} C_DIS
LIN {X -0.039,Y -171.328,Z 1643.379,A 0.000,B 0.000,C 90.000,E1 248.284} C_DIS
LIN {X 0.015,Y -167.583,Z 1643.355,A 0.000,B 0.000,C 90.000,E1 243.948} C_DIS
LIN {X -0.046,Y -166.219,Z 1643.346,A 0.000,B 0.000,C 90.000,E1 242.231} C_DIS
LIN {X -0.058,Y -162.981,Z 1643.326,A 0.000,B 0.000,C 90.000,E1 238.742} C_DIS
LIN {X -0.010,Y -160.897,Z 1643.312,A 0.000,B 0.000,C 90.000,E1 236.087} C_DIS
LIN {X -0.033,Y -157.664,Z 1643.292,A 0.000,B 0.000,C 90.000,E1 232.557} C_DIS
LIN {X -0.094,Y -155.702,Z 1643.277,A 0.000,B 0.000,C 90.000,E1 229.908} C_DIS
LIN {X -0.039,Y -151.966,Z 1643.252,A 0.000,B 0.000,C 90.000,E1 225.405} C_DIS
LIN {X -0.022,Y -150.207,Z 1643.237,A 0.000,B 0.000,C 90.000,E1 222.690} C_DIS
LIN {X -0.007,Y -146.974,Z 1643.212,A 0.000,B 0.000,C 90.000,E1 218.141} C_DIS
LIN {X 0.011,Y -145.560,Z 1643.197,A 0.000,B 0.000,C 90.000,E1 215.391} C_DIS
LIN {X 0.011,Y -142.952,Z 1643.171,A 0.000,B 0.000,C 90.000,E1 210.797} C_DIS
LIN {X -0.058,Y -141.578,Z 1643.151,A 0.000,B 0.000,C 90.000,E1 207.129} C_DIS
LIN {X -0.011,Y -139.415,Z 1643.115,A 0.000,B 0.000,C 90.000,E1 200.610} C_DIS
LIN {X 0.041,Y -139.140,Z 1643.104,A 0.000,B 0.000,C 90.000,E1 198.725} C_DIS
LIN {X 0.068,Y -138.348,Z 1643.057,A 0.000,B 0.000,C 90.000,E1 190.310} C_DIS
LIN {X 0.056,Y -139.492,Z 1643.005,A 0.000,B 0.000,C 90.000,E1 180.974} C_DIS
LIN {X -0.003,Y -141.104,Z 1642.974,A 0.000,B 0.000,C 90.000,E1 175.412} C_DIS
LIN {X -0.050,Y -142.483,Z 1642.959,A 0.000,B 0.000,C 90.000,E1 172.648} C_DIS
LIN {X 0.039,Y -144.733,Z 1642.933,A 0.000,B 0.000,C 90.000,E1 167.993} C_DIS
LIN {X -0.011,Y -147.337,Z 1642.913,A 0.000,B 0.000,C 90.000,E1 164.338} C_DIS
LIN {X 0.055,Y -150.661,Z 1642.888,A 0.000,B 0.000,C 90.000,E1 159.752} C_DIS
LIN {X -0.064,Y -154.140,Z 1642.868,A 0.000,B 0.000,C 90.000,E1 156.177} C_DIS
LIN {X -0.002,Y -157.568,Z 1642.848,A 0.000,B 0.000,C 90.000,E1 152.564} C_DIS
LIN {X 0.022,Y -161.812,Z 1642.828,A 0.000,B 0.000,C 90.000,E1 148.997} C_DIS
LIN {X 0.042,Y -166.004,Z 1642.808,A 0.000,B 0.000,C 90.000,E1 145.468} C_DIS
LIN {X 0.034,Y -171.003,Z 1642.789,A 0.000,B 0.000,C 90.000,E1 141.984} C_DIS
LIN {X -0.050,Y -175.872,Z 1642.770,A 0.000,B 0.000,C 90.000,E1 138.566} C_DIS
LIN {X -0.057,Y -181.477,Z 1642.751,A 0.000,B 0.000,C 90.000,E1 135.162} C_DIS
LIN {X 0.079,Y -186.990,Z 1642.732,A 0.000,B 0.000,C 90.000,E1 131.757} C_DIS
LIN {X 0.081,Y -190.106,Z 1642.723,A 0.000,B 0.000,C 90.000,E1 130.092} C_DIS
LIN {X 0.100,Y -195.878,Z 1642.705,A 0.000,B 0.000,C 90.000,E1 126.790} C_DIS
LIN {X -0.108,Y -200.710,Z 1642.691,A 0.000,B 0.000,C 90.000,E1 124.405} C_DIS
LIN {X -0.006,Y -206.646,Z 1642.673,A 0.000,B 0.000,C 90.000,E1 121.131} C_DIS
LIN {X -0.060,Y -326.933,Z 1642.673,A 0.000,B 0.000,C 90.000,E1 121.131} C_DIS
LIN {X 0.067,Y -328.630,Z 1642.673,A 0.000,B 0.000,C 90.000,E1 121.082} C_DIS
LIN {X -0.091,Y -332.947,Z 1642.672,A 0.000,B 0.000,C 90.000,E1 120.924} C_DIS
LIN {X 0.037,Y -335.376,Z 1642.671,A 0.000,B 0.000,C 90.000,E1 120.718} C_DIS
LIN {X 0.123,Y -338.682,Z 1642.669,A 0.000,B 0.000,C 90.000,E1 120.335} C_DIS
LIN {X 0.040,Y -340.596,Z 1642.667,A 0.000,B 0.000,C 90.000,E1 120.050} C_DIS
LIN {X 0.082,Y -342.091,Z 1642.665,A 0.000,B 0.000,C 90.000,E1 119.745} C_DIS
LIN {X 0.036,Y -354.262,Z 1642.650,A 0.000,B 0.000,C 90.000,E1 117.001} C_DIS
LIN {X -0.159,Y -367.889,Z 1642.635,A 0.000,B 0.000,C 90.000,E1 114.335} C_DIS
LIN {X -0.047,Y -381.327,Z 1642.622,A 0.000,B 0.000,C 90.000,E1 111.972} C_DIS
LIN {X -0.105,Y -396.107,Z 1642.609,A 0.000,B 0.000,C 90.000,E1 109.685} C_DIS
LIN {X 0.185,Y -412.331,Z 1642.597,A 0.000,B 0.000,C 90.000,E1 107.402} C_DIS
LIN {X -0.030,Y -430.113,Z 1642.585,A 0.000,B 0.000,C 90.000,E1 105.245} C_DIS
LIN {X 0.019,Y -449.485,Z 1642.573,A 0.000,B 0.000,C 90.000,E1 103.119} C_DIS
LIN {X 0.203,Y -469.642,Z 1642.562,A 0.000,B 0.000,C 90.000,E1 101.130} C_DIS
LIN {X -0.168,Y -492.927,Z 1642.551,A 0.000,B 0.000,C 90.000,E1 99.151} C_DIS
LIN {X 0.152,Y -498.186,Z 1642.548,A 0.000,B 0.000,C 90.000,E1 98.690} C_DIS
LIN {X -0.124,Y -500.443,Z 1642.547,A 0.000,B 0.000,C 90.000,E1 98.511} C_DIS
LIN {X -0.092,Y -502.302,Z 1642.546,A 0.000,B 0.000,C 90.000,E1 98.276} C_DIS
LIN {X -0.133,Y -503.712,Z 1642.545,A 0.000,B 0.000,C 90.000,E1 98.049} C_DIS
LIN {X 0.167,Y -505.602,Z 1642.542,A 0.000,B 0.000,C 90.000,E1 97.530} C_DIS
LIN {X -0.024,Y -506.351,Z 1642.539,A 0.000,B 0.000,C 90.000,E1 97.068} C_DIS
LIN {X -0.205,Y -506.089,Z 1642.537,A 0.000,B 0.000,C 90.000,E1 96.606} C_DIS
LIN {X 0.120,Y -504.774,Z 1642.534,A 0.000,B 0.000,C 90.000,E1 96.087} C_DIS
LIN {X 0.057,Y -503.654,Z 1642.533,A 0.000,B 0.000,C 90.000,E1 95.853} C_DIS
LIN {X -0.131,Y -500.411,Z 1642.530,A 0.000,B 0.000,C 90.000,E1 95.391} C_DIS
LIN {X -0.142,Y -486.816,Z 1642.519,A 0.000,B 0.000,C 90.000,E1 93.440} C_DIS
LIN {X 0.206,Y -474.675,Z 1642.509,A 0.000,B 0.000,C 90.000,E1 91.661} C_DIS
LIN {X 0.009,Y -463.980,Z 1642.501,A 0.000,B 0.000,C 90.000,E1 90.172} C_DIS
LIN {X 0.096,Y -453.004,Z 1642.492,A 0.000,B 0.000,C 90.000,E1 88.625} C_DIS
LIN {X -0.192,Y -443.537,Z 1642.485,A 0.000,B 0.000,C 90.000,E1 87.364} C_DIS
LIN {X 0.020,Y -431.749,Z 1642.476,A 0.000,B 0.000,C 90.000,E1 85.755} C_DIS
LIN {X 0.018,Y -419.960,Z 1642.468,A 0.000,B 0.000,C 90.000,E1 84.147} C_DIS
LIN {X -0.091,Y -399.089,Z 1642.451,A 0.000,B 0.000,C 90.000,E1 81.141} C_DIS
LIN {X 0.080,Y -381.471,Z 1642.435,A 0.000,B 0.000,C 90.000,E1 78.285} C_DIS
LIN {X -0.103,Y -366.420,Z 1642.420,A 0.000,B 0.000,C 90.000,E1 75.700} C_DIS
LIN {X -0.048,Y -351.940,Z 1642.406,A 0.000,B 0.000,C 90.000,E1 73.015} C_DIS
LIN {X 0.025,Y -335.204,Z 1642.387,A 0.000,B 0.000,C 90.000,E1 69.645} C_DIS
LIN {X 0.113,Y -319.351,Z 1642.368,A 0.000,B 0.000,C 90.000,E1 66.177} C_DIS
LIN {X -0.067,Y -308.567,Z 1642.354,A 0.000,B 0.000,C 90.000,E1 63.640} C_DIS
LIN {X 0.161,Y -299.213,Z 1642.341,A 0.000,B 0.000,C 90.000,E1 61.307} C_DIS
LIN {X 0.072,Y -291.050,Z 1642.330,A 0.000,B 0.000,C 90.000,E1 59.331} C_DIS
LIN {X -0.022,Y -282.676,Z 1642.318,A 0.000,B 0.000,C 90.000,E1 57.327} C_DIS
LIN {X 0.029,Y -274.096,Z 1642.307,A 0.000,B 0.000,C 90.000,E1 55.261} C_DIS
LIN {X -0.006,Y -262.809,Z 1642.292,A 0.000,B 0.000,C 90.000,E1 52.477} C_DIS
LIN {X 0.029,Y -250.613,Z 1642.274,A 0.000,B 0.000,C 90.000,E1 49.256} C_DIS
LIN {X -0.003,Y -239.158,Z 1642.255,A 0.000,B 0.000,C 90.000,E1 45.972} C_DIS
LIN {X -0.010,Y -228.473,Z 1642.237,A 0.000,B 0.000,C 90.000,E1 42.609} C_DIS
LIN {X -0.034,Y -219.675,Z 1642.220,A 0.000,B 0.000,C 90.000,E1 39.564} C_DIS
LIN {X -0.019,Y -211.622,Z 1642.203,A 0.000,B 0.000,C 90.000,E1 36.457} C_DIS
LIN {X 0.013,Y -204.393,Z 1642.185,A 0.000,B 0.000,C 90.000,E1 33.293} C_DIS
LIN {X 0.044,Y -197.890,Z 1642.167,A 0.000,B 0.000,C 90.000,E1 30.079} C_DIS
LIN {X -0.105,Y -192.104,Z 1642.149,A 0.000,B 0.000,C 90.000,E1 26.873} C_DIS
LIN {X -0.058,Y -186.954,Z 1642.131,A 0.000,B 0.000,C 90.000,E1 23.567} C_DIS
LIN {X -0.090,Y -182.511,Z 1642.112,A 0.000,B 0.000,C 90.000,E1 20.248} C_DIS
LIN {X -0.041,Y -177.957,Z 1642.089,A 0.000,B 0.000,C 90.000,E1 16.024} C_DIS
LIN {X -0.034,Y -174.201,Z 1642.065,A 0.000,B 0.000,C 90.000,E1 11.771} C_DIS
LIN {X 0.017,Y -170.825,Z 1642.037,A 0.000,B 0.000,C 90.000,E1 6.606} C_DIS
LIN {X 0.000,Y -168.308,Z 1642.000,A 0.000,B 0.000,C 90.000,E1 360.000} C_DIS
LIN {X 0.017,Y -168.818,Z 1641.935,A 0.000,B 0.000,C 90.000,E1 348.229} C_DIS
LIN {X 0.025,Y -171.541,Z 1641.906,A 0.000,B 0.000,C 90.000,E1 343.032} C_DIS
LIN {X 0.060,Y -175.088,Z 1641.882,A 0.000,B 0.000,C 90.000,E1 338.720} C_DIS
LIN {X -0.098,Y -178.893,Z 1641.863,A 0.000,B 0.000,C 90.000,E1 335.357} C_DIS
LIN {X -0.016,Y -183.598,Z 1641.844,A 0.000,B 0.000,C 90.000,E1 331.948} C_DIS
LIN {X -0.056,Y -189.123,Z 1641.826,A 0.000,B 0.000,C 90.000,E1 328.614} C_DIS
LIN {X -0.052,Y -195.477,Z 1641.807,A 0.000,B 0.000,C 90.000,E1 325.308} C_DIS
LIN {X 0.027,Y -202.756,Z 1641.789,A 0.000,B 0.000,C 90.000,E1 322.029} C_DIS
LIN {X 0.058,Y -209.930,Z 1641.774,A 0.000,B 0.000,C 90.000,E1 319.218} C_DIS
LIN {X 0.135,Y -219.306,Z 1641.756,A 0.000,B 0.000,C 90.000,E1 316.053} C_DIS
LIN {X -0.026,Y -229.879,Z 1641.739,A 0.000,B 0.000,C 90.000,E1 313.014} C_DIS
LIN {X -0.045,Y -240.164,Z 1641.724,A 0.000,B 0.000,C 90.000,E1 310.378} C_DIS
LIN {X -0.122,Y -250.076,Z 1641.712,A 0.000,B 0.000,C 90.000,E1 308.177} C_DIS
LIN {X 0.047,Y -261.103,Z 1641.700,A 0.000,B 0.000,C 90.000,E1 305.964} C_DIS
LIN {X -0.004,Y -275.452,Z 1641.686,A 0.000,B 0.000,C 90.000,E1 303.499} C_DIS
LIN {X 0.071,Y -288.947,Z 1641.675,A 0.000,B 0.000,C 90.000,E1 301.416} C_DIS
LIN {X -0.070,Y -310.952,Z 1641.658,A 0.000,B 0.000,C 90.000,E1 298.437} C_DIS
LIN {X 0.056,Y -323.345,Z 1641.649,A 0.000,B 0.000,C 90.000,E1 296.796} C_DIS
LIN {X 0.080,Y -335.597,Z 1641.640,A 0.000,B 0.000,C 90.000,E1 295.207} C_DIS
LIN {X 0.168,Y -347.654,Z 1641.631,A 0.000,B 0.000,C 90.000,E1 293.643} C_DIS
LIN {X 0.034,Y -362.067,Z 1641.621,A 0.000,B 0.000,C 90.000,E1 291.844} C_DIS
LIN {X 0.059,Y -373.809,Z 1641.613,A 0.000,B 0.000,C 90.000,E1 290.355} C_DIS
LIN {X -0.110,Y -380.468,Z 1641.608,A 0.000,B 0.000,C 90.000,E1 289.504} C_DIS
LIN {X 0.137,Y -386.611,Z 1641.603,A 0.000,B 0.000,C 90.000,E1 288.598} C_DIS
LIN {X -0.037,Y -392.222,Z 1641.599,A 0.000,B 0.000,C 90.000,E1 287.764} C_DIS
LIN {X -0.211,Y -395.546,Z 1641.595,A 0.000,B 0.000,C 90.000,E1 287.221} C_DIS
LIN {X 0.013,Y -398.531,Z 1641.592,A 0.000,B 0.000,C 90.000,E1 286.622} C_DIS
LIN {X -0.054,Y -402.189,Z 1641.588,A 0.000,B 0.000,C 90.000,E1 285.788} C_DIS
LIN {X -0.173,Y -404.154,Z 1641.585,A 0.000,B 0.000,C 90.000,E1 285.245} C_DIS
LIN {X 0.000,Y -405.764,Z 1641.581,A 0.000,B 0.000,C 90.000,E1 284.662} C_DIS
LIN {X -0.104,Y -407.011,Z 1641.578,A 0.000,B 0.000,C 90.000,E1 284.120} C_DIS
LIN {X 0.096,Y -407.838,Z 1641.575,A 0.000,B 0.000,C 90.000,E1 283.536} C_DIS
LIN {X -0.092,Y -408.218,Z 1641.572,A 0.000,B 0.000,C 90.000,E1 283.008} C_DIS
LIN {X 0.214,Y -408.050,Z 1641.569,A 0.000,B 0.000,C 90.000,E1 282.411} C_DIS
LIN {X 0.032,Y -407.440,Z 1641.566,A 0.000,B 0.000,C 90.000,E1 281.883} C_DIS
LIN {X -0.152,Y -406.288,Z 1641.563,A 0.000,B 0.000,C 90.000,E1 281.355} C_DIS
LIN {X -0.017,Y -404.540,Z 1641.560,A 0.000,B 0.000,C 90.000,E1 280.782} C_DIS
LIN {X 0.188,Y -402.128,Z 1641.557,A 0.000,B 0.000,C 90.000,E1 280.197} C_DIS
LIN {X -0.022,Y -399.050,Z 1641.554,A 0.000,B 0.000,C 90.000,E1 279.670} C_DIS
LIN {X 0.081,Y -395.312,Z 1641.551,A 0.000,B 0.000,C 90.000,E1 279.095} C_DIS
LIN {X -0.105,Y -388.866,Z 1641.546,A 0.000,B 0.000,C 90.000,E1 278.276} C_DIS
LIN {X -0.015,Y -381.788,Z 1641.541,A 0.000,B 0.000,C 90.000,E1 277.409} C_DIS
LIN {X -0.007,Y -376.429,Z 1641.538,A 0.000,B 0.000,C 90.000,E1 276.834} C_DIS
LIN {X 0.146,Y -370.691,Z 1641.535,A 0.000,B 0.000,C 90.000,E1 276.258} C_DIS
LIN {X -0.153,Y -364.747,Z 1641.532,A 0.000,B 0.000,C 90.000,E1 275.796} C_DIS
LIN {X 0.138,Y -358.382,Z 1641.529,A 0.000,B 0.000,C 90.000,E1 275.277} C_DIS
LIN {X 0.017,Y -352.057,Z 1641.527,A 0.000,B 0.000,C 90.000,E1 274.878} C_DIS
LIN {X 0.134,Y -345.620,Z 1641.525,A 0.000,B 0.000,C 90.000,E1 274.473} C_DIS
LIN {X 0.128,Y -336.036,Z 1641.522,A 0.000,B 0.000,C 90.000,E1 273.955} C_DIS
LIN {X -0.001,Y -326.116,Z 1641.519,A 0.000,B 0.000,C 90.000,E1 273.498} C_DIS
LIN {X -0.073,Y -316.236,Z 1641.517,A 0.000,B 0.000,C 90.000,E1 273.094} C_DIS
LIN {X 0.120,Y -305.940,Z 1641.515,A 0.000,B 0.000,C 90.000,E1 272.694} C_DIS
LIN {X 0.019,Y -295.201,Z 1641.513,A 0.000,B 0.000,C 90.000,E1 272.407} C_DIS
LIN {X -0.079,Y -283.784,Z 1641.512,A 0.000,B 0.000,C 90.000,E1 272.178} C_DIS
LIN {X 0.105,Y -273.857,Z 1641.511,A 0.000,B 0.000,C 90.000,E1 272.007} C_DIS
LIN {X 0.091,Y -244.696,Z 1641.510,A 0.000,B 0.000,C 90.000,E1 271.776} C_DIS
LIN {X -0.064,Y -222.553,Z 1641.509,A 0.000,B 0.000,C 90.000,E1 271.661} C_DIS
LIN {X -0.001,Y -191.785,Z 1641.509,A 0.000,B 0.000,C 90.000,E1 271.547} C_DIS
LIN {X -0.025,Y -181.343,Z 1641.509,A 0.000,B 0.000,C 90.000,E1 271.547} C_DIS
LIN {X 0.005,Y -181.561,Z 1641.500,A 0.000,B 0.000,C 90.000,E1 270.000} C_DIS
LIN {X -0.039,Y -180.903,Z 1641.474,A 0.000,B 0.000,C 90.000,E1 265.298} C_DIS
LIN {X -0.089,Y -180.238,Z 1641.464,A 0.000,B 0.000,C 90.000,E1 263.628} C_DIS
LIN {X -0.069,Y -178.724,Z 1641.441,A 0.000,B 0.000,C 90.000,E1 259.398} C_DIS
LIN {X -0.001,Y -175.771,Z 1641.413,A 0.000,B 0.000,C 90.000,E1 254.283} C_DIS
LIN {X -0.013,Y -171.955,Z 1641.384,A 0.000,B 0.000,C 90.000,E1 249.156} C_DIS
LIN {X 0.024,Y -171.347,Z 1641.379,A 0.000,B 0.000,C 90.000,E1 248.284} C_DIS
LIN {X 0.002,Y -167.599,Z 1641.355,A 0.000,B 0.000,C 90.000,E1 243.973} C_DIS
LIN {X 0.014,Y -166.241,Z 1641.346,A 0.000,B 0.000,C 90.000,E1 242.231} C_DIS
LIN {X 0.002,Y -162.999,Z 1641.326,A 0.000,B 0.000,C 90.000,E1 238.742} C_DIS
LIN {X 0.049,Y -160.918,Z 1641.312,A 0.000,B 0.000,C 90.000,E1 236.087} C_DIS
LIN {X 0.026,Y -157.682,Z 1641.292,A 0.000,B 0.000,C 90.000,E1 232.557} C_DIS
LIN {X -0.035,Y -155.721,Z 1641.277,A 0.000,B 0.000,C 90.000,E1 229.908} C_DIS
LIN {X 0.018,Y -151.981,Z 1641.252,A 0.000,B 0.000,C 90.000,E1 225.405} C_DIS
LIN {X 0.035,Y -150.224,Z 1641.237,A 0.000,B 0.000,C 90.000,E1 222.690} C_DIS
LIN {X -0.042,Y -146.987,Z 1641.212,A 0.000,B 0.000,C 90.000,E1 218.177} C_DIS
LIN {X -0.051,Y -145.572,Z 1641.197,A 0.000,B 0.000,C 90.000,E1 215.438} C_DIS
LIN {X 0.066,Y -142.963,Z 1641.171,A 0.000,B 0.000,C 90.000,E1 210.797} C_DIS
LIN {X -0.003,Y -141.590,Z 1641.151,A 0.000,B 0.000,C 90.000,E1 207.129} C_DIS
LIN {X 0.043,Y -139.419,Z 1641.115,A 0.000,B 0.000,C 90.000,E1 200.610} C_DIS
LIN {X -0.036,Y -139.146,Z 1641.104,A 0.000,B 0.000,C 90.000,E1 198.779} C_DIS
LIN {X -0.013,Y -138.347,Z 1641.058,A 0.000,B 0.000,C 90.000,E1 190.366} C_DIS
LIN {X -0.028,Y -139.489,Z 1641.006,A 0.000,B 0.000,C 90.000,E1 181.031} C_DIS
LIN {X 0.052,Y -141.095,Z 1640.975,A 0.000,B 0.000,C 90.000,E1 175.412} C_DIS
LIN {X 0.005,Y -142.473,Z 1640.959,A 0.000,B 0.000,C 90.000,E1 172.648} C_DIS
LIN {X -0.046,Y -144.719,Z 1640.933,A 0.000,B 0.000,C 90.000,E1 168.049} C_DIS
LIN {X 0.047,Y -147.320,Z 1640.913,A 0.000,B 0.000,C 90.000,E1 164.338} C_DIS
LIN {X -0.029,Y -150.642,Z 1640.888,A 0.000,B 0.000,C 90.000,E1 159.806} C_DIS
LIN {X -0.006,Y -154.120,Z 1640.868,A 0.000,B 0.000,C 90.000,E1 156.177} C_DIS
LIN {X -0.083,Y -157.545,Z 1640.848,A 0.000,B 0.000,C 90.000,E1 152.615} C_DIS
LIN {X 0.083,Y -161.784,Z 1640.828,A 0.000,B 0.000,C 90.000,E1 148.997} C_DIS
LIN {X -0.034,Y -165.976,Z 1640.808,A 0.000,B 0.000,C 90.000,E1 145.515} C_DIS
LIN {X -0.038,Y -170.971,Z 1640.789,A 0.000,B 0.000,C 90.000,E1 142.029} C_DIS
LIN {X 0.013,Y -175.840,Z 1640.770,A 0.000,B 0.000,C 90.000,E1 138.566} C_DIS
LIN {X 0.008,Y -181.446,Z 1640.751,A 0.000,B 0.000,C 90.000,E1 135.162} C_DIS
LIN {X -0.119,Y -186.954,Z 1640.732,A 0.000,B 0.000,C 90.000,E1 131.838} C_DIS
LIN {X 0.002,Y -190.068,Z 1640.723,A 0.000,B 0.000,C 90.000,E1 130.135} C_DIS
LIN {X -0.106,Y -195.842,Z 1640.705,A 0.000,B 0.000,C 90.000,E1 126.870} C_DIS
LIN {X -0.039,Y -200.674,Z 1640.691,A 0.000,B 0.000,C 90.000,E1 124.405} C_DIS
LIN {X -0.046,Y -206.571,Z 1640.673,A 0.000,B 0.000,C 90.000,E1 121.180} C_DIS
LIN {X 0.173,Y -326.662,Z 1640.673,A 0.000,B 0.000,C 90.000,E1 121.131} C_DIS
LIN {X -0.104,Y -329.223,Z 1640.673,A 0.000,B 0.000,C 90.000,E1 121.131} C_DIS
LIN {X 0.022,Y -333.082,Z 1640.672,A 0.000,B 0.000,C 90.000,E1 120.924} C_DIS
LIN {X -0.023,Y -335.419,Z 1640.671,A 0.000,B 0.000,C 90.000,E1 120.747} C_DIS
LIN {X -0.056,Y -338.645,Z 1640.669,A 0.000,B 0.000,C 90.000,E1 120.384} C_DIS
LIN {X -0.047,Y -340.553,Z 1640.667,A 0.000,B 0.000,C 90.000,E1 120.079} C_DIS
LIN {X -0.007,Y -343.325,Z 1640.664,A 0.000,B 0.000,C 90.000,E1 119.461} C_DIS
LIN {X -0.199,Y -355.639,Z 1640.648,A 0.000,B 0.000,C 90.000,E1 116.744} C_DIS
LIN {X -0.021,Y -369.426,Z 1640.633,A 0.000,B 0.000,C 90.000,E1 114.027} C_DIS
LIN {X 0.137,Y -383.021,Z 1640.620,A 0.000,B 0.000,C 90.000,E1 111.663} C_DIS
LIN {X -0.005,Y -397.971,Z 1640.608,A 0.000,B 0.000,C 90.000,E1 109.396} C_DIS
LIN {X -0.048,Y -414.377,Z 1640.595,A 0.000,B 0.000,C 90.000,E1 107.166} C_DIS
LIN {X 0.196,Y -432.355,Z 1640.583,A 0.000,B 0.000,C 90.000,E1 104.954} C_DIS
LIN {X -0.065,Y -451.864,Z 1640.572,A 0.000,B 0.000,C 90.000,E1 102.883} C_DIS
LIN {X -0.185,Y -472.088,Z 1640.561,A 0.000,B 0.000,C 90.000,E1 100.950} C_DIS
LIN {X 0.058,Y -495.468,Z 1640.550,A 0.000,B 0.000,C 90.000,E1 98.916} C_DIS
LIN {X 0.200,Y -498.086,Z 1640.548,A 0.000,B 0.000,C 90.000,E1 98.690} C_DIS
LIN {X -0.077,Y -500.321,Z 1640.547,A 0.000,B 0.000,C 90.000,E1 98.511} C_DIS
LIN {X -0.058,Y -502.175,Z 1640.546,A 0.000,B 0.000,C 90.000,E1 98.276} C_DIS
LIN {X -0.111,Y -503.578,Z 1640.545,A 0.000,B 0.000,C 90.000,E1 98.049} C_DIS
LIN {X 0.189,Y -505.446,Z 1640.542,A 0.000,B 0.000,C 90.000,E1 97.530} C_DIS
LIN {X -0.004,Y -506.175,Z 1640.539,A 0.000,B 0.000,C 90.000,E1 97.068} C_DIS
LIN {X -0.185,Y -505.894,Z 1640.537,A 0.000,B 0.000,C 90.000,E1 96.606} C_DIS
LIN {X 0.139,Y -504.558,Z 1640.534,A 0.000,B 0.000,C 90.000,E1 96.087} C_DIS
LIN {X 0.075,Y -503.427,Z 1640.533,A 0.000,B 0.000,C 90.000,E1 95.853} C_DIS
LIN {X -0.114,Y -500.176,Z 1640.530,A 0.000,B 0.000,C 90.000,E1 95.391} C_DIS
LIN {X -0.131,Y -486.593,Z 1640.519,A 0.000,B 0.000,C 90.000,E1 93.440} C_DIS
LIN {X 0.213,Y -474.482,Z 1640.509,A 0.000,B 0.000,C 90.000,E1 91.661} C_DIS
LIN {X 0.012,Y -463.775,Z 1640.501,A 0.000,B 0.000,C 90.000,E1 90.172} C_DIS
LIN {X 0.096,Y -452.821,Z 1640.492,A 0.000,B 0.000,C 90.000,E1 88.625} C_DIS
LIN {X -0.194,Y -443.354,Z 1640.485,A 0.000,B 0.000,C 90.000,E1 87.364} C_DIS
LIN {X 0.013,Y -431.538,Z 1640.476,A 0.000,B 0.000,C 90.000,E1 85.755} C_DIS
LIN {X 0.008,Y -419.718,Z 1640.468,A 0.000,B 0.000,C 90.000,E1 84.147} C_DIS
LIN {X -0.108,Y -398.814,Z 1640.451,A 0.000,B 0.000,C 90.000,E1 81.141} C_DIS
LIN {X 0.056,Y -381.205,Z 1640.435,A 0.000,B 0.000,C 90.000,E1 78.285} C_DIS
LIN {X -0.132,Y -366.176,Z 1640.420,A 0.000,B 0.000,C 90.000,E1 75.700} C_DIS
LIN {X -0.084,Y -351.691,Z 1640.406,A 0.000,B 0.000,C 90.000,E1 73.015} C_DIS
LIN {X -0.016,Y -334.969,Z 1640.387,A 0.000,B 0.000,C 90.000,E1 69.645} C_DIS
LIN {X 0.065,Y -319.102,Z 1640.368,A 0.000,B 0.000,C 90.000,E1 66.177} C_DIS
LIN {X -0.119,Y -308.352,Z 1640.353,A 0.000,B 0.000,C 90.000,E1 63.640} C_DIS
LIN {X 0.107,Y -299.012,Z 1640.341,A 0.000,B 0.000,C 90.000,E1 61.307} C_DIS
LIN {X 0.015,Y -290.882,Z 1640.330,A 0.000,B 0.000,C 90.000,E1 59.331} C_DIS
LIN {X -0.080,Y -282.536,Z 1640.318,A 0.000,B 0.000,C 90.000,E1 57.327} C_DIS
LIN {X -0.030,Y -273.947,Z 1640.307,A 0.000,B 0.000,C 90.000,E1 55.261} C_DIS
LIN {X -0.066,Y -262.644,Z 1640.292,A 0.000,B 0.000,C 90.000,E1 52.477} C_DIS
LIN {X -0.033,Y -250.422,Z 1640.274,A 0.000,B 0.000,C 90.000,E1 49.256} C_DIS
LIN {X -0.067,Y -238.916,Z 1640.255,A 0.000,B 0.000,C 90.000,E1 45.972} C_DIS
LIN {X -0.078,Y -228.226,Z 1640.237,A 0.000,B 0.000,C 90.000,E1 42.609} C_DIS
LIN {X -0.106,Y -219.449,Z 1640.220,A 0.000,B 0.000,C 90.000,E1 39.564} C_DIS
LIN {X 0.031,Y -211.389,Z 1640.202,A 0.000,B 0.000,C 90.000,E1 36.423} C_DIS
LIN {X -0.066,Y -204.212,Z 1640.185,A 0.000,B 0.000,C 90.000,E1 33.293} C_DIS
LIN {X -0.037,Y -197.733,Z 1640.167,A 0.000,B 0.000,C 90.000,E1 30.079} C_DIS
LIN {X -0.015,Y -192.013,Z 1640.149,A 0.000,B 0.000,C 90.000,E1 26.821} C_DIS
LIN {X 0.033,Y -186.896,Z 1640.131,A 0.000,B 0.000,C 90.000,E1 23.515} C_DIS
LIN {X 0.064,Y -182.503,Z 1640.112,A 0.000,B 0.000,C 90.000,E1 20.174} C_DIS
LIN {X 0.052,Y -177.967,Z 1640.089,A 0.000,B 0.000,C 90.000,E1 15.969} C_DIS
LIN {X 0.062,Y -174.253,Z 1640.065,A 0.000,B 0.000,C 90.000,E1 11.715} C_DIS
LIN {X -0.056,Y -170.882,Z 1640.037,A 0.000,B 0.000,C 90.000,E1 6.606} C_DIS
LIN {X -0.031,Y -168.301,Z 1639.997,A 0.000,B 0.000,C 90.000,E1 359.542} C_DIS
LIN {X 0.025,Y -168.935,Z 1639.935,A 0.000,B 0.000,C 90.000,E1 348.229} C_DIS
LIN {X 0.037,Y -171.663,Z 1639.906,A 0.000,B 0.000,C 90.000,E1 343.032} C_DIS
LIN {X 0.077,Y -175.204,Z 1639.882,A 0.000,B 0.000,C 90.000,E1 338.720} C_DIS
LIN {X -0.078,Y -179.035,Z 1639.863,A 0.000,B 0.000,C 90.000,E1 335.357} C_DIS
LIN {X -0.079,Y -183.748,Z 1639.844,A 0.000,B 0.000,C 90.000,E1 331.975} C_DIS
LIN {X -0.028,Y -189.303,Z 1639.826,A 0.000,B 0.000,C 90.000,E1 328.614} C_DIS
LIN {X -0.018,Y -195.661,Z 1639.807,A 0.000,B 0.000,C 90.000,E1 325.308} C_DIS
LIN {X -0.057,Y -202.934,Z 1639.789,A 0.000,B 0.000,C 90.000,E1 322.065} C_DIS
LIN {X -0.034,Y -210.079,Z 1639.774,A 0.000,B 0.000,C 90.000,E1 319.256} C_DIS
LIN {X -0.123,Y -219.435,Z 1639.756,A 0.000,B 0.000,C 90.000,E1 316.134} C_DIS
LIN {X 0.031,Y -229.971,Z 1639.739,A 0.000,B 0.000,C 90.000,E1 313.014} C_DIS
LIN {X 0.017,Y -240.218,Z 1639.724,A 0.000,B 0.000,C 90.000,E1 310.378} C_DIS
LIN {X -0.057,Y -250.099,Z 1639.712,A 0.000,B 0.000,C 90.000,E1 308.177} C_DIS
LIN {X -0.096,Y -261.123,Z 1639.700,A 0.000,B 0.000,C 90.000,E1 306.011} C_DIS
LIN {X 0.068,Y -275.431,Z 1639.686,A 0.000,B 0.000,C 90.000,E1 303.499} C_DIS
LIN {X -0.135,Y -291.297,Z 1639.673,A 0.000,B 0.000,C 90.000,E1 301.131} C_DIS
LIN {X 0.010,Y -310.945,Z 1639.658,A 0.000,B 0.000,C 90.000,E1 298.437} C_DIS
LIN {X -0.006,Y -323.323,Z 1639.649,A 0.000,B 0.000,C 90.000,E1 296.821} C_DIS
LIN {X 0.167,Y -335.596,Z 1639.640,A 0.000,B 0.000,C 90.000,E1 295.207} C_DIS
LIN {X -0.054,Y -350.032,Z 1639.630,A 0.000,B 0.000,C 90.000,E1 293.387} C_DIS
LIN {X 0.127,Y -362.042,Z 1639.621,A 0.000,B 0.000,C 90.000,E1 291.844} C_DIS
LIN {X 0.025,Y -373.786,Z 1639.613,A 0.000,B 0.000,C 90.000,E1 290.375} C_DIS
LIN {X -0.013,Y -380.455,Z 1639.608,A 0.000,B 0.000,C 90.000,E1 289.504} C_DIS
LIN {X -0.131,Y -386.612,Z 1639.604,A 0.000,B 0.000,C 90.000,E1 288.652} C_DIS
LIN {X 0.064,Y -392.260,Z 1639.599,A 0.000,B 0.000,C 90.000,E1 287.764} C_DIS
LIN {X 0.055,Y -397.127,Z 1639.594,A 0.000,B 0.000,C 90.000,E1 286.913} C_DIS
LIN {X -0.023,Y -401.150,Z 1639.589,A 0.000,B 0.000,C 90.000,E1 286.079} C_DIS
LIN {X -0.068,Y -404.308,Z 1639.585,A 0.000,B 0.000,C 90.000,E1 285.245} C_DIS
LIN {X 0.106,Y -405.950,Z 1639.582,A 0.000,B 0.000,C 90.000,E1 284.662} C_DIS
LIN {X 0.002,Y -407.235,Z 1639.578,A 0.000,B 0.000,C 90.000,E1 284.120} C_DIS
LIN {X -0.193,Y -408.084,Z 1639.575,A 0.000,B 0.000,C 90.000,E1 283.592} C_DIS
LIN {X 0.018,Y -408.473,Z 1639.572,A 0.000,B 0.000,C 90.000,E1 283.008} C_DIS
LIN {X -0.162,Y -408.399,Z 1639.569,A 0.000,B 0.000,C 90.000,E1 282.479} C_DIS
LIN {X 0.060,Y -407.798,Z 1639.566,A 0.000,B 0.000,C 90.000,E1 281.895} C_DIS
LIN {X -0.118,Y -406.663,Z 1639.563,A 0.000,B 0.000,C 90.000,E1 281.366} C_DIS
LIN {X 0.099,Y -404.945,Z 1639.560,A 0.000,B 0.000,C 90.000,E1 280.782} C_DIS
LIN {X -0.091,Y -402.570,Z 1639.557,A 0.000,B 0.000,C 90.000,E1 280.254} C_DIS
LIN {X 0.097,Y -399.502,Z 1639.554,A 0.000,B 0.000,C 90.000,E1 279.670} C_DIS
LIN {X -0.191,Y -395.792,Z 1639.551,A 0.000,B 0.000,C 90.000,E1 279.151} C_DIS
LIN {X 0.017,Y -389.319,Z 1639.546,A 0.000,B 0.000,C 90.000,E1 278.276} C_DIS
LIN {X 0.109,Y -382.206,Z 1639.541,A 0.000,B 0.000,C 90.000,E1 277.409} C_DIS
LIN {X 0.191,Y -376.960,Z 1639.538,A 0.000,B 0.000,C 90.000,E1 276.834} C_DIS
LIN {X -0.022,Y -371.241,Z 1639.535,A 0.000,B 0.000,C 90.000,E1 276.315} C_DIS
LIN {X 0.027,Y -365.221,Z 1639.532,A 0.000,B 0.000,C 90.000,E1 275.796} C_DIS
LIN {X -0.001,Y -358.968,Z 1639.530,A 0.000,B 0.000,C 90.000,E1 275.334} C_DIS
LIN {X -0.143,Y -352.591,Z 1639.527,A 0.000,B 0.000,C 90.000,E1 274.935} C_DIS
LIN {X 0.002,Y -346.248,Z 1639.525,A 0.000,B 0.000,C 90.000,E1 274.531} C_DIS
LIN {X -0.008,Y -336.608,Z 1639.522,A 0.000,B 0.000,C 90.000,E1 274.012} C_DIS
LIN {X -0.102,Y -326.873,Z 1639.520,A 0.000,B 0.000,C 90.000,E1 273.555} C_DIS
LIN {X 0.120,Y -316.922,Z 1639.517,A 0.000,B 0.000,C 90.000,E1 273.094} C_DIS
LIN {X -0.010,Y -306.579,Z 1639.515,A 0.000,B 0.000,C 90.000,E1 272.751} C_DIS
LIN {X -0.088,Y -296.124,Z 1639.514,A 0.000,B 0.000,C 90.000,E1 272.465} C_DIS
LIN {X -0.091,Y -288.821,Z 1639.513,A 0.000,B 0.000,C 90.000,E1 272.293} C_DIS
LIN {X 0.021,Y -280.820,Z 1639.512,A 0.000,B 0.000,C 90.000,E1 272.121} C_DIS
LIN {X -0.009,Y -269.781,Z 1639.511,A 0.000,B 0.000,C 90.000,E1 272.007} C_DIS
LIN {X 0.003,Y -239.986,Z 1639.510,A 0.000,B 0.000,C 90.000,E1 271.776} C_DIS
LIN {X -0.058,Y -220.355,Z 1639.509,A 0.000,B 0.000,C 90.000,E1 271.661} C_DIS
LIN {X 0.049,Y -190.570,Z 1639.509,A 0.000,B 0.000,C 90.000,E1 271.547} C_DIS
LIN {X 0.025,Y -181.341,Z 1639.509,A 0.000,B 0.000,C 90.000,E1 271.547} C_DIS
LIN {X -0.074,Y -181.566,Z 1639.500,A 0.000,B 0.000,C 90.000,E1 270.057} C_DIS
LIN {X 0.064,Y -180.905,Z 1639.474,A 0.000,B 0.000,C 90.000,E1 265.298} C_DIS
LIN {X 0.015,Y -180.253,Z 1639.465,A 0.000,B 0.000,C 90.000,E1 263.628} C_DIS
LIN {X 0.033,Y -178.743,Z 1639.441,A 0.000,B 0.000,C 90.000,E1 259.398} C_DIS
LIN {X -0.069,Y -175.791,Z 1639.413,A 0.000,B 0.000,C 90.000,E1 254.338} C_DIS
LIN {X -0.074,Y -171.975,Z 1639.384,A 0.000,B 0.000,C 90.000,E1 249.209} C_DIS
LIN {X -0.036,Y -171.378,Z 1639.380,A 0.000,B 0.000,C 90.000,E1 248.337} C_DIS
LIN {X -0.051,Y -167.624,Z 1639.356,A 0.000,B 0.000,C 90.000,E1 244.024} C_DIS
LIN {X -0.036,Y -166.276,Z 1639.346,A 0.000,B 0.000,C 90.000,E1 242.281} C_DIS
LIN {X -0.041,Y -163.027,Z 1639.327,A 0.000,B 0.000,C 90.000,E1 238.791} C_DIS
LIN {X 0.011,Y -160.954,Z 1639.312,A 0.000,B 0.000,C 90.000,E1 236.135} C_DIS
LIN {X -0.004,Y -157.709,Z 1639.292,A 0.000,B 0.000,C 90.000,E1 232.603} C_DIS
LIN {X 0.058,Y -155.748,Z 1639.277,A 0.000,B 0.000,C 90.000,E1 229.908} C_DIS
LIN {X 0.004,Y -152.005,Z 1639.252,A 0.000,B 0.000,C 90.000,E1 225.445} C_DIS
LIN {X -0.086,Y -150.251,Z 1639.237,A 0.000,B 0.000,C 90.000,E1 222.771} C_DIS
LIN {X 0.049,Y -147.008,Z 1639.212,A 0.000,B 0.000,C 90.000,E1 218.177} C_DIS
LIN {X 0.038,Y -145.592,Z 1639.197,A 0.000,B 0.000,C 90.000,E1 215.438} C_DIS
LIN {X -0.041,Y -142.979,Z 1639.171,A 0.000,B 0.000,C 90.000,E1 210.875} C_DIS
LIN {X -0.041,Y -141.606,Z 1639.151,A 0.000,B 0.000,C 90.000,E1 207.180} C_DIS
LIN {X 0.000,Y -139.425,Z 1639.115,A 0.000,B 0.000,C 90.000,E1 200.663} C_DIS
LIN {X 0.051,Y -139.154,Z 1639.104,A 0.000,B 0.000,C 90.000,E1 198.779} C_DIS
LIN {X 0.073,Y -138.344,Z 1639.058,A 0.000,B 0.000,C 90.000,E1 190.366} C_DIS
LIN {X 0.060,Y -139.484,Z 1639.006,A 0.000,B 0.000,C 90.000,E1 181.031} C_DIS
LIN {X 0.000,Y -141.079,Z 1638.975,A 0.000,B 0.000,C 90.000,E1 175.469} C_DIS
LIN {X -0.046,Y -142.455,Z 1638.959,A 0.000,B 0.000,C 90.000,E1 172.704} C_DIS
LIN {X 0.043,Y -144.698,Z 1638.934,A 0.000,B 0.000,C 90.000,E1 168.049} C_DIS
LIN {X -0.004,Y -147.293,Z 1638.913,A 0.000,B 0.000,C 90.000,E1 164.393} C_DIS
LIN {X 0.012,Y -150.612,Z 1638.888,A 0.000,B 0.000,C 90.000,E1 159.826} C_DIS
LIN {X -0.053,Y -154.087,Z 1638.868,A 0.000,B 0.000,C 90.000,E1 156.230} C_DIS
LIN {X 0.013,Y -157.508,Z 1638.848,A 0.000,B 0.000,C 90.000,E1 152.615} C_DIS
LIN {X -0.042,Y -161.739,Z 1638.828,A 0.000,B 0.000,C 90.000,E1 149.076} C_DIS
LIN {X 0.064,Y -165.932,Z 1638.809,A 0.000,B 0.000,C 90.000,E1 145.515} C_DIS
LIN {X -0.043,Y -170.921,Z 1638.789,A 0.000,B 0.000,C 90.000,E1 142.065} C_DIS
LIN {X -0.017,Y -175.789,Z 1638.770,A 0.000,B 0.000,C 90.000,E1 138.609} C_DIS
LIN {X -0.017,Y -181.397,Z 1638.751,A 0.000,B 0.000,C 90.000,E1 135.202} C_DIS
LIN {X -0.014,Y -186.896,Z 1638.732,A 0.000,B 0.000,C 90.000,E1 131.838} C_DIS
LIN {X -0.061,Y -191.478,Z 1638.719,A 0.000,B 0.000,C 90.000,E1 129.358} C_DIS
LIN {X -0.130,Y -197.337,Z 1638.700,A 0.000,B 0.000,C 90.000,E1 126.091} C_DIS
LIN {X 0.071,Y -200.614,Z 1638.691,A 0.000,B 0.000,C 90.000,E1 124.405} C_DIS
LIN {X 0.015,Y -206.479,Z 1638.673,A 0.000,B 0.000,C 90.000,E1 121.209} C_DIS
LIN {X -0.029,Y -326.145,Z 1638.673,A 0.000,B 0.000,C 90.000,E1 121.209} C_DIS
LIN {X -0.112,Y -330.218,Z 1638.673,A 0.000,B 0.000,C 90.000,E1 121.131} C_DIS
LIN {X 0.086,Y -333.319,Z 1638.672,A 0.000,B 0.000,C 90.000,E1 120.924} C_DIS
LIN {X 0.063,Y -336.993,Z 1638.670,A 0.000,B 0.000,C 90.000,E1 120.590} C_DIS
LIN {X 0.022,Y -340.521,Z 1638.667,A 0.000,B 0.000,C 90.000,E1 120.079} C_DIS
LIN {X 0.011,Y -343.290,Z 1638.664,A 0.000,B 0.000,C 90.000,E1 119.461} C_DIS
LIN {X -0.175,Y -355.599,Z 1638.648,A 0.000,B 0.000,C 90.000,E1 116.744} C_DIS
LIN {X -0.003,Y -369.389,Z 1638.633,A 0.000,B 0.000,C 90.000,E1 114.027} C_DIS
LIN {X -0.201,Y -382.981,Z 1638.620,A 0.000,B 0.000,C 90.000,E1 111.716} C_DIS
LIN {X 0.011,Y -397.928,Z 1638.608,A 0.000,B 0.000,C 90.000,E1 109.396} C_DIS
LIN {X -0.032,Y -414.334,Z 1638.595,A 0.000,B 0.000,C 90.000,E1 107.166} C_DIS
LIN {X -0.206,Y -432.310,Z 1638.583,A 0.000,B 0.000,C 90.000,E1 105.009} C_DIS
LIN {X -0.053,Y -451.822,Z 1638.572,A 0.000,B 0.000,C 90.000,E1 102.883} C_DIS
LIN {X -0.175,Y -472.045,Z 1638.561,A 0.000,B 0.000,C 90.000,E1 100.950} C_DIS
LIN {X 0.086,Y -495.397,Z 1638.550,A 0.000,B 0.000,C 90.000,E1 98.916} C_DIS
LIN {X 0.209,Y -498.039,Z 1638.548,A 0.000,B 0.000,C 90.000,E1 98.690} C_DIS
LIN {X -0.074,Y -500.246,Z 1638.547,A 0.000,B 0.000,C 90.000,E1 98.511} C_DIS
LIN {X 0.136,Y -501.923,Z 1638.546,A 0.000,B 0.000,C 90.000,E1 98.276} C_DIS
LIN {X -0.006,Y -503.397,Z 1638.545,A 0.000,B 0.000,C 90.000,E1 98.049} C_DIS
LIN {X -0.078,Y -504.490,Z 1638.543,A 0.000,B 0.000,C 90.000,E1 97.814} C_DIS
LIN {X 0.228,Y -505.756,Z 1638.541,A 0.000,B 0.000,C 90.000,E1 97.296} C_DIS
LIN {X 0.039,Y -505.975,Z 1638.538,A 0.000,B 0.000,C 90.000,E1 96.834} C_DIS
LIN {X -0.144,Y -505.184,Z 1638.535,A 0.000,B 0.000,C 90.000,E1 96.372} C_DIS
LIN {X 0.176,Y -503.244,Z 1638.533,A 0.000,B 0.000,C 90.000,E1 95.853} C_DIS
LIN {X -0.010,Y -500.014,Z 1638.530,A 0.000,B 0.000,C 90.000,E1 95.391} C_DIS
LIN {X 0.113,Y -488.167,Z 1638.521,A 0.000,B 0.000,C 90.000,E1 93.669} C_DIS
LIN {X 0.156,Y -477.833,Z 1638.512,A 0.000,B 0.000,C 90.000,E1 92.178} C_DIS
LIN {X 0.026,Y -467.247,Z 1638.504,A 0.000,B 0.000,C 90.000,E1 90.688} C_DIS
LIN {X 0.171,Y -456.388,Z 1638.495,A 0.000,B 0.000,C 90.000,E1 89.141} C_DIS
LIN {X -0.065,Y -447.087,Z 1638.488,A 0.000,B 0.000,C 90.000,E1 87.879} C_DIS
LIN {X 0.012,Y -437.370,Z 1638.481,A 0.000,B 0.000,C 90.000,E1 86.560} C_DIS
LIN {X -0.030,Y -421.548,Z 1638.469,A 0.000,B 0.000,C 90.000,E1 84.432} C_DIS
LIN {X -0.137,Y -400.477,Z 1638.452,A 0.000,B 0.000,C 90.000,E1 81.432} C_DIS
LIN {X 0.107,Y -381.004,Z 1638.435,A 0.000,B 0.000,C 90.000,E1 78.285} C_DIS
LIN {X -0.084,Y -366.011,Z 1638.421,A 0.000,B 0.000,C 90.000,E1 75.700} C_DIS
LIN {X -0.046,Y -351.504,Z 1638.406,A 0.000,B 0.000,C 90.000,E1 73.015} C_DIS
LIN {X 0.138,Y -336.293,Z 1638.389,A 0.000,B 0.000,C 90.000,E1 69.934} C_DIS
LIN {X -0.103,Y -321.661,Z 1638.371,A 0.000,B 0.000,C 90.000,E1 66.847} C_DIS
LIN {X -0.100,Y -308.198,Z 1638.353,A 0.000,B 0.000,C 90.000,E1 63.640} C_DIS
LIN {X 0.125,Y -298.886,Z 1638.341,A 0.000,B 0.000,C 90.000,E1 61.307} C_DIS
LIN {X 0.030,Y -290.778,Z 1638.330,A 0.000,B 0.000,C 90.000,E1 59.331} C_DIS
LIN {X -0.067,Y -282.458,Z 1638.318,A 0.000,B 0.000,C 90.000,E1 57.327} C_DIS
LIN {X -0.018,Y -273.864,Z 1638.307,A 0.000,B 0.000,C 90.000,E1 55.261} C_DIS
LIN {X -0.125,Y -263.924,Z 1638.293,A 0.000,B 0.000,C 90.000,E1 52.844} C_DIS
LIN {X -0.054,Y -251.596,Z 1638.276,A 0.000,B 0.000,C 90.000,E1 49.622} C_DIS
LIN {X 0.121,Y -239.966,Z 1638.257,A 0.000,B 0.000,C 90.000,E1 46.296} C_DIS
LIN {X -0.038,Y -229.171,Z 1638.239,A 0.000,B 0.000,C 90.000,E1 42.975} C_DIS
LIN {X -0.054,Y -220.298,Z 1638.222,A 0.000,B 0.000,C 90.000,E1 39.930} C_DIS
LIN {X 0.103,Y -212.175,Z 1638.205,A 0.000,B 0.000,C 90.000,E1 36.790} C_DIS
LIN {X 0.026,Y -204.935,Z 1638.187,A 0.000,B 0.000,C 90.000,E1 33.658} C_DIS
LIN {X 0.007,Y -198.392,Z 1638.169,A 0.000,B 0.000,C 90.000,E1 30.463} C_DIS
LIN {X 0.040,Y -192.628,Z 1638.151,A 0.000,B 0.000,C 90.000,E1 27.206} C_DIS
LIN {X -0.070,Y -187.459,Z 1638.133,A 0.000,B 0.000,C 90.000,E1 23.951} C_DIS
LIN {X -0.019,Y -183.020,Z 1638.115,A 0.000,B 0.000,C 90.000,E1 20.610} C_DIS
LIN {X 0.043,Y -178.432,Z 1638.091,A 0.000,B 0.000,C 90.000,E1 16.386} C_DIS
LIN {X -0.065,Y -174.652,Z 1638.068,A 0.000,B 0.000,C 90.000,E1 12.175} C_DIS
LIN {X 0.019,Y -171.189,Z 1638.039,A 0.000,B 0.000,C 90.000,E1 7.004} C_DIS
LIN {X 0.000,Y -168.517,Z 1638.000,A 0.000,B 0.000,C 90.000,E1 360.000} C_DIS
LIN {X 0.008,Y -168.739,Z 1637.939,A 0.000,B 0.000,C 90.000,E1 349.106} C_DIS
LIN {X -0.026,Y -171.241,Z 1637.911,A 0.000,B 0.000,C 90.000,E1 343.921} C_DIS
LIN {X -0.053,Y -174.515,Z 1637.887,A 0.000,B 0.000,C 90.000,E1 339.625} C_DIS
LIN {X 0.038,Y -178.124,Z 1637.868,A 0.000,B 0.000,C 90.000,E1 336.177} C_DIS
LIN {X 0.019,Y -182.650,Z 1637.849,A 0.000,B 0.000,C 90.000,E1 332.794} C_DIS
LIN {X -0.041,Y -188.027,Z 1637.830,A 0.000,B 0.000,C 90.000,E1 329.459} C_DIS
LIN {X -0.001,Y -194.163,Z 1637.812,A 0.000,B 0.000,C 90.000,E1 326.135} C_DIS
LIN {X 0.089,Y -201.230,Z 1637.794,A 0.000,B 0.000,C 90.000,E1 322.844} C_DIS
LIN {X -0.055,Y -208.095,Z 1637.778,A 0.000,B 0.000,C 90.000,E1 320.070} C_DIS
LIN {X -0.034,Y -217.120,Z 1637.760,A 0.000,B 0.000,C 90.000,E1 316.905} C_DIS
LIN {X 0.060,Y -227.327,Z 1637.743,A 0.000,B 0.000,C 90.000,E1 313.785} C_DIS
LIN {X -0.013,Y -237.232,Z 1637.729,A 0.000,B 0.000,C 90.000,E1 311.148} C_DIS
LIN {X 0.011,Y -246.719,Z 1637.716,A 0.000,B 0.000,C 90.000,E1 308.910} C_DIS
LIN {X 0.065,Y -257.342,Z 1637.704,A 0.000,B 0.000,C 90.000,E1 306.710} C_DIS
LIN {X -0.144,Y -269.121,Z 1637.692,A 0.000,B 0.000,C 90.000,E1 304.612} C_DIS
LIN {X 0.101,Y -282.012,Z 1637.681,A 0.000,B 0.000,C 90.000,E1 302.467} C_DIS
LIN {X -0.094,Y -303.407,Z 1637.664,A 0.000,B 0.000,C 90.000,E1 299.461} C_DIS
LIN {X 0.179,Y -315.932,Z 1637.654,A 0.000,B 0.000,C 90.000,E1 297.769} C_DIS
LIN {X 0.188,Y -330.739,Z 1637.644,A 0.000,B 0.000,C 90.000,E1 295.848} C_DIS
LIN {X -0.108,Y -342.806,Z 1637.635,A 0.000,B 0.000,C 90.000,E1 294.335} C_DIS
LIN {X 0.125,Y -357.226,Z 1637.625,A 0.000,B 0.000,C 90.000,E1 292.461} C_DIS
LIN {X 0.079,Y -369.121,Z 1637.617,A 0.000,B 0.000,C 90.000,E1 290.972} C_DIS
LIN {X -0.030,Y -378.257,Z 1637.610,A 0.000,B 0.000,C 90.000,E1 289.812} C_DIS
LIN {X -0.159,Y -384.630,Z 1637.605,A 0.000,B 0.000,C 90.000,E1 288.960} C_DIS
LIN {X 0.129,Y -390.452,Z 1637.600,A 0.000,B 0.000,C 90.000,E1 288.055} C_DIS
LIN {X -0.008,Y -395.654,Z 1637.596,A 0.000,B 0.000,C 90.000,E1 287.221} C_DIS
LIN {X -0.103,Y -399.997,Z 1637.591,A 0.000,B 0.000,C 90.000,E1 286.386} C_DIS
LIN {X -0.152,Y -403.496,Z 1637.586,A 0.000,B 0.000,C 90.000,E1 285.552} C_DIS
LIN {X -0.173,Y -406.135,Z 1637.582,A 0.000,B 0.000,C 90.000,E1 284.717} C_DIS
LIN {X 0.117,Y -407.473,Z 1637.578,A 0.000,B 0.000,C 90.000,E1 284.120} C_DIS
LIN {X -0.077,Y -408.375,Z 1637.575,A 0.000,B 0.000,C 90.000,E1 283.592} C_DIS
LIN {X 0.136,Y -408.759,Z 1637.572,A 0.000,B 0.000,C 90.000,E1 283.008} C_DIS
LIN {X -0.043,Y -408.748,Z 1637.569,A 0.000,B 0.000,C 90.000,E1 282.479} C_DIS
LIN {X -0.219,Y -408.164,Z 1637.566,A 0.000,B 0.000,C 90.000,E1 281.951} C_DIS
LIN {X 0.004,Y -407.066,Z 1637.563,A 0.000,B 0.000,C 90.000,E1 281.366} C_DIS
LIN {X -0.175,Y -405.380,Z 1637.560,A 0.000,B 0.000,C 90.000,E1 280.838} C_DIS
LIN {X 0.035,Y -403.031,Z 1637.557,A 0.000,B 0.000,C 90.000,E1 280.254} C_DIS
LIN {X -0.169,Y -400.014,Z 1637.554,A 0.000,B 0.000,C 90.000,E1 279.726} C_DIS
LIN {X -0.061,Y -396.327,Z 1637.551,A 0.000,B 0.000,C 90.000,E1 279.151} C_DIS
LIN {X 0.149,Y -389.896,Z 1637.546,A 0.000,B 0.000,C 90.000,E1 278.276} C_DIS
LIN {X -0.135,Y -382.725,Z 1637.541,A 0.000,B 0.000,C 90.000,E1 277.466} C_DIS
LIN {X -0.122,Y -377.316,Z 1637.538,A 0.000,B 0.000,C 90.000,E1 276.891} C_DIS
LIN {X 0.049,Y -371.571,Z 1637.535,A 0.000,B 0.000,C 90.000,E1 276.315} C_DIS
LIN {X 0.087,Y -365.506,Z 1637.532,A 0.000,B 0.000,C 90.000,E1 275.796} C_DIS
LIN {X 0.177,Y -356.191,Z 1637.529,A 0.000,B 0.000,C 90.000,E1 275.106} C_DIS
LIN {X 0.093,Y -346.535,Z 1637.525,A 0.000,B 0.000,C 90.000,E1 274.531} C_DIS
LIN {X 0.077,Y -336.843,Z 1637.522,A 0.000,B 0.000,C 90.000,E1 274.012} C_DIS
LIN {X -0.009,Y -327.059,Z 1637.520,A 0.000,B 0.000,C 90.000,E1 273.555} C_DIS
LIN {X -0.100,Y -317.163,Z 1637.517,A 0.000,B 0.000,C 90.000,E1 273.151} C_DIS
LIN {X 0.064,Y -306.699,Z 1637.515,A 0.000,B 0.000,C 90.000,E1 272.751} C_DIS
LIN {X -0.131,Y -299.791,Z 1637.514,A 0.000,B 0.000,C 90.000,E1 272.579} C_DIS
LIN {X -0.012,Y -288.948,Z 1637.513,A 0.000,B 0.000,C 90.000,E1 272.293} C_DIS
LIN {X 0.097,Y -280.898,Z 1637.512,A 0.000,B 0.000,C 90.000,E1 272.121} C_DIS
LIN {X 0.083,Y -263.902,Z 1637.511,A 0.000,B 0.000,C 90.000,E1 271.949} C_DIS
LIN {X -0.052,Y -229.349,Z 1637.510,A 0.000,B 0.000,C 90.000,E1 271.718} C_DIS
LIN {X 0.067,Y -211.190,Z 1637.509,A 0.000,B 0.000,C 90.000,E1 271.604} C_DIS
LIN {X -0.075,Y -191.864,Z 1637.509,A 0.000,B 0.000,C 90.000,E1 271.604} C_DIS
LIN {X 0.087,Y -181.336,Z 1637.509,A 0.000,B 0.000,C 90.000,E1 271.547} C_DIS
LIN {X -0.058,Y -181.566,Z 1637.500,A 0.000,B 0.000,C 90.000,E1 270.057} C_DIS
LIN {X 0.080,Y -180.905,Z 1637.474,A 0.000,B 0.000,C 90.000,E1 265.298} C_DIS
LIN {X 0.030,Y -180.255,Z 1637.465,A 0.000,B 0.000,C 90.000,E1 263.628} C_DIS
LIN {X 0.048,Y -178.747,Z 1637.441,A 0.000,B 0.000,C 90.000,E1 259.398} C_DIS
LIN {X -0.054,Y -175.794,Z 1637.413,A 0.000,B 0.000,C 90.000,E1 254.338} C_DIS
LIN {X -0.059,Y -171.978,Z 1637.384,A 0.000,B 0.000,C 90.000,E1 249.209} C_DIS
LIN {X -0.021,Y -171.382,Z 1637.380,A 0.000,B 0.000,C 90.000,E1 248.337} C_DIS
LIN {X -0.035,Y -167.627,Z 1637.356,A 0.000,B 0.000,C 90.000,E1 244.024} C_DIS
LIN {X -0.020,Y -166.281,Z 1637.346,A 0.000,B 0.000,C 90.000,E1 242.281} C_DIS
LIN {X -0.026,Y -163.030,Z 1637.327,A 0.000,B 0.000,C 90.000,E1 238.791} C_DIS
LIN {X 0.026,Y -160.959,Z 1637.312,A 0.000,B 0.000,C 90.000,E1 236.135} C_DIS
LIN {X 0.010,Y -157.713,Z 1637.292,A 0.000,B 0.000,C 90.000,E1 232.603} C_DIS
LIN {X 0.073,Y -155.753,Z 1637.277,A 0.000,B 0.000,C 90.000,E1 229.908} C_DIS
LIN {X 0.018,Y -152.009,Z 1637.253,A 0.000,B 0.000,C 90.000,E1 225.445} C_DIS
LIN {X -0.072,Y -150.255,Z 1637.237,A 0.000,B 0.000,C 90.000,E1 222.771} C_DIS
LIN {X 0.063,Y -147.011,Z 1637.212,A 0.000,B 0.000,C 90.000,E1 218.177} C_DIS
LIN {X 0.052,Y -145.594,Z 1637.197,A 0.000,B 0.000,C 90.000,E1 215.438} C_DIS
LIN {X -0.028,Y -142.981,Z 1637.172,A 0.000,B 0.000,C 90.000,E1 210.875} C_DIS
LIN {X -0.027,Y -141.608,Z 1637.151,A 0.000,B 0.000,C 90.000,E1 207.180} C_DIS
LIN {X 0.014,Y -139.426,Z 1637.115,A 0.000,B 0.000,C 90.000,E1 200.663} C_DIS
LIN {X 0.064,Y -139.155,Z 1637.104,A 0.000,B 0.000,C 90.000,E1 198.779} C_DIS
LIN {X -0.049,Y -138.344,Z 1637.058,A 0.000,B 0.000,C 90.000,E1 190.423} C_DIS
LIN {X -0.067,Y -139.483,Z 1637.006,A 0.000,B 0.000,C 90.000,E1 181.088} C_DIS
LIN {X 0.014,Y -141.077,Z 1636.975,A 0.000,B 0.000,C 90.000,E1 175.469} C_DIS
LIN {X -0.033,Y -142.452,Z 1636.959,A 0.000,B 0.000,C 90.000,E1 172.704} C_DIS
LIN {X 0.057,Y -144.694,Z 1636.934,A 0.000,B 0.000,C 90.000,E1 168.049} C_DIS
LIN {X 0.009,Y -147.289,Z 1636.913,A 0.000,B 0.000,C 90.000,E1 164.393} C_DIS
LIN {X 0.025,Y -150.608,Z 1636.888,A 0.000,B 0.000,C 90.000,E1 159.826} C_DIS
LIN {X -0.039,Y -154.082,Z 1636.868,A 0.000,B 0.000,C 90.000,E1 156.230} C_DIS
LIN {X 0.027,Y -157.503,Z 1636.848,A 0.000,B 0.000,C 90.000,E1 152.615} C_DIS
LIN {X -0.028,Y -161.732,Z 1636.828,A 0.000,B 0.000,C 90.000,E1 149.076} C_DIS
LIN {X -0.015,Y -165.925,Z 1636.809,A 0.000,B 0.000,C 90.000,E1 145.548} C_DIS
LIN {X -0.028,Y -170.913,Z 1636.789,A 0.000,B 0.000,C 90.000,E1 142.065} C_DIS
LIN {X -0.002,Y -175.782,Z 1636.770,A 0.000,B 0.000,C 90.000,E1 138.609} C_DIS
LIN {X -0.001,Y -181.390,Z 1636.751,A 0.000,B 0.000,C 90.000,E1 135.202} C_DIS
LIN {X 0.002,Y -186.888,Z 1636.732,A 0.000,B 0.000,C 90.000,E1 131.838} C_DIS
LIN {X -0.045,Y -191.470,Z 1636.719,A 0.000,B 0.000,C 90.000,E1 129.358} C_DIS
LIN {X -0.113,Y -197.328,Z 1636.700,A 0.000,B 0.000,C 90.000,E1 126.091} C_DIS
LIN {X 0.088,Y -200.605,Z 1636.691,A 0.000,B 0.000,C 90.000,E1 124.405} C_DIS
LIN {X -0.016,Y -206.399,Z 1636.674,A 0.000,B 0.000,C 90.000,E1 121.258} C_DIS
LIN {X -0.089,Y -326.479,Z 1636.674,A 0.000,B 0.000,C 90.000,E1 121.258} C_DIS
LIN {X -0.003,Y -328.377,Z 1636.673,A 0.000,B 0.000,C 90.000,E1 121.209} C_DIS
LIN {X 0.089,Y -331.789,Z 1636.673,A 0.000,B 0.000,C 90.000,E1 121.052} C_DIS
